// TIA Portal project "Project_Benzinarie" (V15.1)

(* hardware
DEVICE "S71500/ET200MP station_1"  S7-1500 station
   slot 0: "Rail_0"  Rack  6ES7 590-1***0-0AA0
   slot 1: "PLC_1"  CPU 1513-1 PN  6ES7 513-1AL02-0AB0  V2.6
      slot 3: "CPU display_1"  6ES7591-1AA00-0AA0
DEVICE "HMI_1"  KTP900 Basic PN
   slot 0: "HMI_1"  KTP900 Basic PN  6AV2 123-2JB03-0AX0  15.1.0.0
   slot 1: "HMI_RT_1"  KTP900 Basic PN  6AV2 123-2JB03-0AX0  15.1.0.0
   slot 5: "HMI_1.IE_CP_1"  PROFINET Interface  15.0.1.0
      slot 1: "PROFINET Interface_1"  PROFINET Interface
         slot 1: "Port_1"  Port
*)

// ===== PLC "PLC_1"  CPU 1513-1 PN =====

VAR_GLOBAL   // PLC tag table "Default tag table"
   "Clock_Byte" AT %MB0 : Byte;
   "Clock_10Hz" AT %M0.0 : Bool;
   "Clock_5Hz" AT %M0.1 : Bool;
   "Clock_2.5Hz" AT %M0.2 : Bool;
   "Clock_2Hz" AT %M0.3 : Bool;
   "Clock_1.25Hz" AT %M0.4 : Bool;
   "Clock_1Hz" AT %M0.5 : Bool;
   "Clock_0.625Hz" AT %M0.6 : Bool;
   "Clock_0.5Hz" AT %M0.7 : Bool;
END_VAR

DATA_BLOCK "Alarme"   // DB1
{ S7_Optimized_Access := 'TRUE' }
VERSION : 0.1
   VAR
      alarme_gather : Word;
      alarme_vect : Array[0..15] of Bool;
   END_VAR
BEGIN
END_DATA_BLOCK

DATA_BLOCK "Avarii"   // DB2
{ S7_Optimized_Access := 'TRUE' }
VERSION : 0.1
   VAR
      esd : Bool;
      esd_btn : Bool;
      reset_esd : Bool;
      avarie_p1 : Bool;
      avarie_p2 : Bool;
      avarie_p3 : Bool;
      avarie_p4 : Bool;
      avarie_generala : Bool;
      reset_avarii : Bool;
      plata_general : Bool;
   END_VAR
BEGIN
END_DATA_BLOCK

DATA_BLOCK "Bazine"   // DB3
{ S7_Optimized_Access := 'TRUE' }
VERSION : 0.1
   VAR
      benzina_90 : Real;
      benzina_95 : Real;
      motorina : Real;
      motorina_premium : Real;
      "benzina_90_1/2" : Real;
      "benzina_95_1/2" : Real;
      "motorina_1/2" : Real;
      "motorina_premium_1/2" : Real;
      b90_gol : Bool;
      b95_gol : Bool;
      m_gol : Bool;
      m_p_gol : Bool;
      bazin_gol_general : Bool;
      nivel_benzina90 : Real;
      nivel_benzina95 : Real;
      nivel_motorina : Real;
      nivel_motorina_premium : Real;
   END_VAR
BEGIN
END_DATA_BLOCK

DATA_BLOCK "Pompa_benzian90"   // DB4
{ S7_Optimized_Access := 'TRUE' }
VERSION : 0.1
   VAR
      blocare : Bool;
      scoasa : Bool;
      start_clapeta : Bool;
      buton_plata : Bool;
      led_rosu : Bool;
      permisiune_start : Bool;
      index_pret : Real;
      cantitate : Real;
      plata_posibila : Bool;
      terminat : Bool;
      pret : Real;
      nivel_pompa : Real;
      permisiune_pompa : Bool;
      pune_inapoi : Bool;
   END_VAR
BEGIN
END_DATA_BLOCK

DATA_BLOCK "Pompa_benzina95"   // DB5
{ S7_Optimized_Access := 'TRUE' }
VERSION : 0.1
   VAR
      blocare : Bool;
      scoasa : Bool;
      start_clapeta : Bool;
      buton_plata : Bool;
      led_rosu : Bool;
      permisiune_start : Bool;
      index_pret : Real;
      cantitate : Real;
      plata_posibila : Bool;
      terminat : Bool;
      pret : Real;
      nivel_pompa : Real;
      permisiune_pompa : Bool;
      pune_inapoi : Bool;
   END_VAR
BEGIN
END_DATA_BLOCK

DATA_BLOCK "Pompa_motorina"   // DB6
{ S7_Optimized_Access := 'TRUE' }
VERSION : 0.1
   VAR
      blocare : Bool;
      scoasa : Bool;
      start_clapeta : Bool;
      buton_plata : Bool;
      led_rosu : Bool;
      permisiune_start : Bool;
      index_pret : Real;
      cantitate : Real;
      plata_posibila : Bool;
      terminat : Bool;
      pret : Real;
      nivel_pompa : Real;
      permisiune_pompa : Bool;
      pune_inapoi : Bool;
   END_VAR
BEGIN
END_DATA_BLOCK

DATA_BLOCK "Pompa_motorina_premium"   // DB7
{ S7_Optimized_Access := 'TRUE' }
VERSION : 0.1
   VAR
      blocare : Bool;
      scoasa : Bool;
      start_clapeta : Bool;
      buton_plata : Bool;
      led_rosu : Bool;
      permisiune_start : Bool;
      index_pret : Real;
      cantitate : Real;
      plata_posibila : Bool;
      terminat : Bool;
      pret : Real;
      nivel_pompa : Real;
      permisiune_pompa : Bool;
      pune_inapoi : Bool;
   END_VAR
BEGIN
END_DATA_BLOCK

DATA_BLOCK "Benzina90"   // DB8
{ S7_Optimized_Access := 'TRUE' }
VERSION : 0.1
// stored: InstanceOfName Pompa
"Pompa"
BEGIN
END_DATA_BLOCK

DATA_BLOCK "Benzina95"   // DB9
{ S7_Optimized_Access := 'TRUE' }
VERSION : 0.1
// stored: InstanceOfName Pompa
"Pompa"
BEGIN
END_DATA_BLOCK

DATA_BLOCK "Motorina"   // DB10
{ S7_Optimized_Access := 'TRUE' }
VERSION : 0.1
// stored: InstanceOfName Pompa
"Pompa"
BEGIN
END_DATA_BLOCK

DATA_BLOCK "Motorina_premium"   // DB11
{ S7_Optimized_Access := 'TRUE' }
VERSION : 0.1
// stored: InstanceOfName Pompa
"Pompa"
BEGIN
END_DATA_BLOCK

DATA_BLOCK "Butoane_umplere_bazine"   // DB13
{ S7_Optimized_Access := 'TRUE' }
VERSION : 0.1
   VAR
      btn_b90 : Bool;
      btn_b95 : Bool;
      btn_m : Bool;
      btn_m_p : Bool;
   END_VAR
BEGIN
END_DATA_BLOCK

DATA_BLOCK "Hysteresis_DB"   // DB16
{ S7_Optimized_Access := 'TRUE' }
VERSION : 0.1
// stored: InstanceOfName Hysteresis
"Hysteresis"
BEGIN
END_DATA_BLOCK

// folder: System blocks/Program resources

DATA_BLOCK "reset_esd"   // DB12
{ S7_Optimized_Access := 'TRUE' }
AUTHOR : Simatic
FAMILY : IEC
NAME : IEC_TMR
VERSION : 1.0
// stored: InstanceOfName IEC_TIMER
"IEC_TIMER"
BEGIN
END_DATA_BLOCK

DATA_BLOCK "reset_avarii"   // DB14
{ S7_Optimized_Access := 'TRUE' }
AUTHOR : Simatic
FAMILY : IEC
NAME : IEC_TMR
VERSION : 1.0
// stored: InstanceOfName IEC_TIMER
"IEC_TIMER"
BEGIN
END_DATA_BLOCK

DATA_BLOCK "reset_umplere_b90"   // DB17
{ S7_Optimized_Access := 'TRUE' }
AUTHOR : Simatic
FAMILY : IEC
NAME : IEC_TMR
VERSION : 1.0
// stored: InstanceOfName IEC_TIMER
"IEC_TIMER"
BEGIN
END_DATA_BLOCK

DATA_BLOCK "reset_umplere_b95"   // DB18
{ S7_Optimized_Access := 'TRUE' }
AUTHOR : Simatic
FAMILY : IEC
NAME : IEC_TMR
VERSION : 1.0
// stored: InstanceOfName IEC_TIMER
"IEC_TIMER"
BEGIN
END_DATA_BLOCK

DATA_BLOCK "reset_umplere_m"   // DB19
{ S7_Optimized_Access := 'TRUE' }
AUTHOR : Simatic
FAMILY : IEC
NAME : IEC_TMR
VERSION : 1.0
// stored: InstanceOfName IEC_TIMER
"IEC_TIMER"
BEGIN
END_DATA_BLOCK

DATA_BLOCK "reset_umplere_m_p"   // DB20
{ S7_Optimized_Access := 'TRUE' }
AUTHOR : Simatic
FAMILY : IEC
NAME : IEC_TMR
VERSION : 1.0
// stored: InstanceOfName IEC_TIMER
"IEC_TIMER"
BEGIN
END_DATA_BLOCK

// folder: (top level)

FUNCTION_BLOCK "Pompa"   // FB1, LAD
{ S7_Optimized_Access := 'TRUE' }
VERSION : 0.1
   VAR_INPUT
      blocare : Bool;
      esd : Bool;
      avarie_interna : Bool;
      bazin_gol : Bool;
   END_VAR
   VAR_OUTPUT
      pret : Real;
      terminat : Bool;
   END_VAR
   VAR_IN_OUT
      scoasa : Bool;
      start_clapeta : Bool;
      bazin : Real;
      buton_plata : Bool;
      led_rosu : Bool;
      permisiune_start : Bool;
      permisiune_pompa : Bool;
      pune_inapoi : Bool;
      index_pret : Real;
      cantitate : Real;
      plata_posibila : Bool;
      nivel_pompa : Real;
   END_VAR
   VAR
      re1 : Bool;
      re2 : Bool;
      re3 : Bool;
      led_intermitent : Bool;
      timer_reset_plata : TON_TIME;
      Hysteresis_Instance : "Hysteresis";
   END_VAR
   VAR_TEMP   // added for the SCL form of the ladder/FBD networks
      _w1 : Bool;
   END_VAR
BEGIN

REGION Network 1: permisiune de start
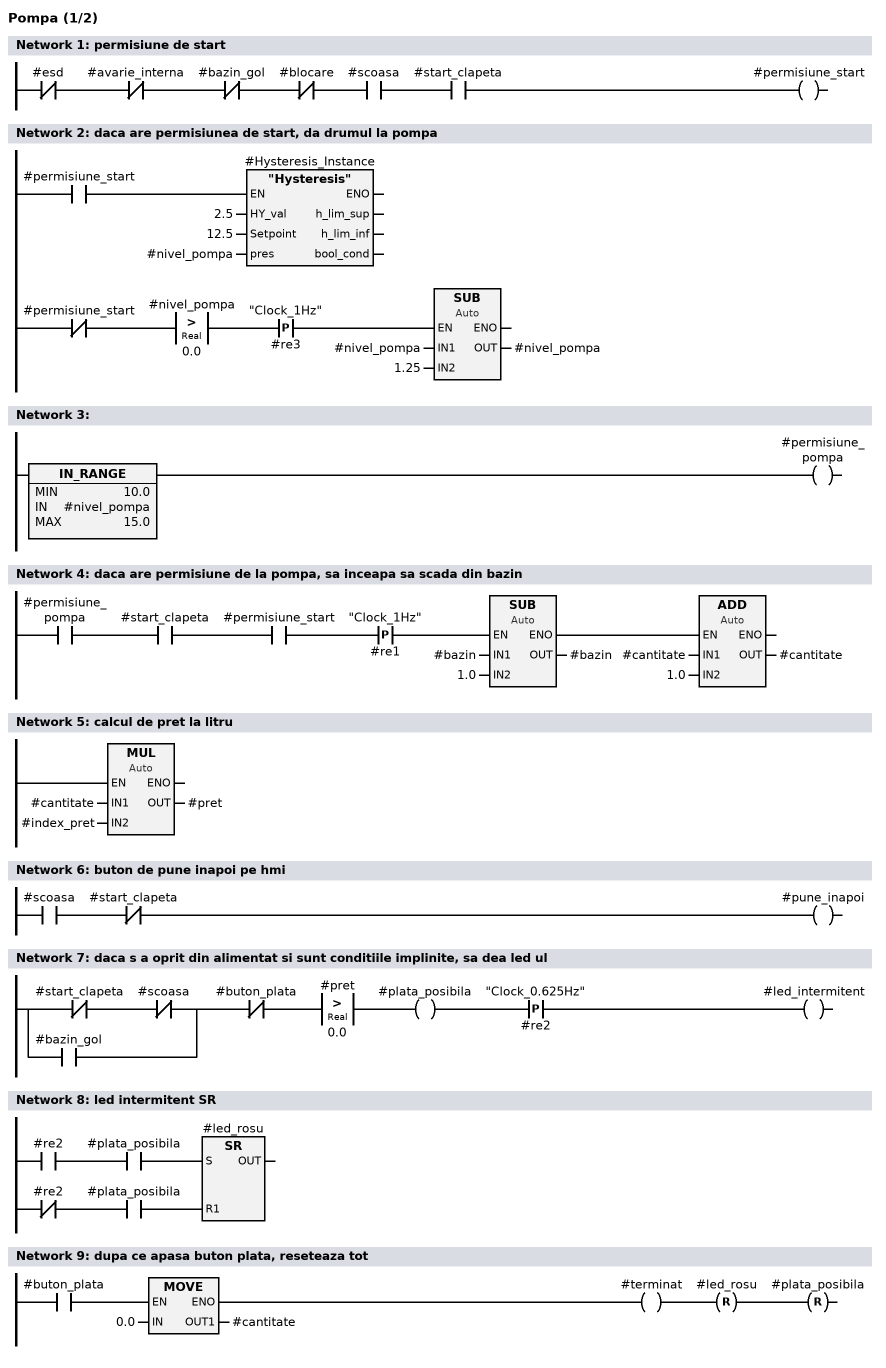
   RUNG wire#powerrail
      I_Contact( #esd )
      I_Contact( #avarie_interna )
      I_Contact( #bazin_gol )
      I_Contact( #blocare )
      Contact( #scoasa )
      Contact( #start_clapeta )
      Coil( #permisiune_start )
   END_RUNG
   // the same network as SCL:
   #permisiune_start := NOT #esd AND NOT #avarie_interna AND NOT #bazin_gol AND NOT #blocare AND #scoasa AND #start_clapeta;
END_REGION

REGION Network 2: daca are permisiunea de start, da drumul la pompa
   RUNG wire#powerrail
      Contact( #permisiune_start )
      #Hysteresis_Instance(HY_val := 2.5, Setpoint := 12.5, pres := #nivel_pompa, h_lim_sup =>, h_lim_inf =>, bool_cond =>)
   END_RUNG
   RUNG wire#powerrail
      I_Contact( #permisiune_start )
      { S7_Templates := "SrcType := Real" } GT_Contact(in1 := #nivel_pompa, in2 := 0.0)
      P_Contact(operand := "Clock_1Hz", bit := #re3)
      Sub(in1 := #nivel_pompa, in2 := 1.25, out => #nivel_pompa)
   END_RUNG
   // the same network as SCL:
   IF #permisiune_start THEN
       #Hysteresis_Instance(HY_val := 2.5, Setpoint := 12.5, pres := #nivel_pompa);   // "Hysteresis"
   END_IF;
   #_w1 := NOT #permisiune_start AND (#nivel_pompa > 0.0) AND "Clock_1Hz" AND NOT #re3;   // rising edge of "Clock_1Hz"
   #re3 := "Clock_1Hz";
   IF #_w1 THEN #nivel_pompa := #nivel_pompa - 1.25; END_IF;
END_REGION

REGION Network 3
   RUNG wire#powerrail
      { S7_Templates := "SrcType := Real" } InRange(min := 10.0, in := #nivel_pompa, max := 15.0)
      Coil( #permisiune_pompa )
   END_RUNG
   // the same network as SCL:
   #permisiune_pompa := (10.0 <= #nivel_pompa) AND (#nivel_pompa <= 15.0);
END_REGION

REGION Network 4: daca are permisiune de la pompa, sa inceapa sa scada din bazin
   RUNG wire#powerrail
      Contact( #permisiune_pompa )
      Contact( #start_clapeta )
      Contact( #permisiune_start )
      P_Contact(operand := "Clock_1Hz", bit := #re1)
      Sub(in1 := #bazin, in2 := 1.0, out => #bazin)
      Add(in1 := #cantitate, in2 := 1.0, out => #cantitate)
   END_RUNG
   // the same network as SCL:
   #_w1 := #permisiune_pompa AND #start_clapeta AND #permisiune_start AND "Clock_1Hz" AND NOT #re1;   // rising edge of "Clock_1Hz"
   #re1 := "Clock_1Hz";
   IF #_w1 THEN
       #bazin := #bazin - 1.0;
       #cantitate := #cantitate + 1.0;
   END_IF;
END_REGION

REGION Network 5: calcul de pret la litru
   RUNG wire#powerrail
      Mul(in1 := #cantitate, in2 := #index_pret, out => #pret)
   END_RUNG
   // the same network as SCL:
   #pret := #cantitate * #index_pret;
END_REGION

REGION Network 6: buton de pune inapoi pe hmi
   RUNG wire#powerrail
      Contact( #scoasa )
      I_Contact( #start_clapeta )
      Coil( #pune_inapoi )
   END_RUNG
   // the same network as SCL:
   #pune_inapoi := #scoasa AND NOT #start_clapeta;
END_REGION

REGION Network 7: daca s a oprit din alimentat si sunt conditiile implinite, sa dea led ul
   RUNG wire#powerrail
      I_Contact( #start_clapeta )
      I_Contact( #scoasa )
      wire#w1
      I_Contact( #buton_plata )
      { S7_Templates := "SrcType := Real" } GT_Contact(in1 := #pret, in2 := 0.0)
      Coil( #plata_posibila )
      P_Contact(operand := "Clock_0.625Hz", bit := #re2)
      Coil( #led_intermitent )
   END_RUNG
   RUNG wire#powerrail
      Contact( #bazin_gol )
   END_RUNG wire#w1
   // the same network as SCL:
   #plata_posibila := ((NOT #start_clapeta AND NOT #scoasa) OR #bazin_gol) AND NOT #buton_plata AND (#pret > 0.0);
   #_w1 := #plata_posibila AND "Clock_0.625Hz" AND NOT #re2;   // rising edge of "Clock_0.625Hz"
   #re2 := "Clock_0.625Hz";
   #led_intermitent := #_w1;
END_REGION

REGION Network 8: led intermitent SR
   RUNG wire#powerrail
      Contact( #re2 )
      Contact( #plata_posibila )
      S_SR(operand := #led_rosu, r1 := wire#w1)
   END_RUNG
   RUNG wire#powerrail
      I_Contact( #re2 )
      Contact( #plata_posibila )
   END_RUNG wire#w1
   // the same network as SCL:
   IF #re2 AND #plata_posibila THEN
       #led_rosu := TRUE;   // SR flip-flop
   END_IF;
   IF NOT #re2 AND #plata_posibila THEN #led_rosu := FALSE; END_IF;
END_REGION

REGION Network 9: dupa ce apasa buton plata, reseteaza tot
   RUNG wire#powerrail
      Contact( #buton_plata )
      Move(in := 0.0, out1 => #cantitate)
      Coil( #terminat )
      R_Coil( #led_rosu )
      R_Coil( #plata_posibila )
   END_RUNG
   // the same network as SCL:
   IF #buton_plata THEN #cantitate := 0.0; END_IF;
   #terminat := #buton_plata;
   IF #buton_plata THEN
       #led_rosu := FALSE;
       #plata_posibila := FALSE;
   END_IF;
END_REGION

REGION Network 10: reseteaza buton plata dupa 3 secunde
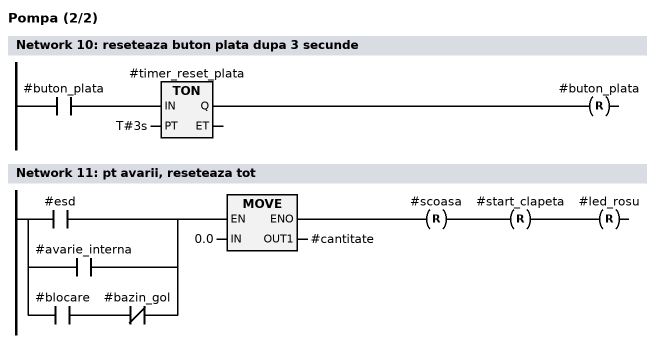
   #timer_reset_plata(IN := #buton_plata, PT := T#3s);   // TON
   IF #timer_reset_plata.Q THEN #buton_plata := FALSE; END_IF;
END_REGION

REGION Network 11: pt avarii, reseteaza tot
   RUNG wire#powerrail
      Contact( #esd )
      wire#w1
      Move(in := 0.0, out1 => #cantitate)
      R_Coil( #scoasa )
      R_Coil( #start_clapeta )
      R_Coil( #led_rosu )
   END_RUNG
   RUNG wire#powerrail
      Contact( #avarie_interna )
   END_RUNG wire#w1
   RUNG wire#powerrail
      Contact( #blocare )
      I_Contact( #bazin_gol )
   END_RUNG wire#w1
   // the same network as SCL:
   IF #esd OR #avarie_interna OR (#blocare AND NOT #bazin_gol) THEN
       #cantitate := 0.0;
       #scoasa := FALSE;
       #start_clapeta := FALSE;
       #led_rosu := FALSE;
   END_IF;
END_REGION
END_FUNCTION_BLOCK

FUNCTION_BLOCK "Hysteresis"   // FB2, LAD
{ S7_Optimized_Access := 'TRUE' }
VERSION : 0.1
   VAR_INPUT
      HY_val : Real;
      Setpoint : Real;
   END_VAR
   VAR_OUTPUT
      h_lim_sup : Real;
      h_lim_inf : Real;
      bool_cond : Bool;
   END_VAR
   VAR_IN_OUT
      pres : Real;
   END_VAR
   VAR
      re1 : Bool;
      re2 : Bool;
      urcare : Bool;
   END_VAR
   VAR_TEMP   // added for the SCL form of the ladder/FBD networks
      _w1 : Bool;
   END_VAR
BEGIN

REGION Network 1: daca are comanda de bool, sa creasca
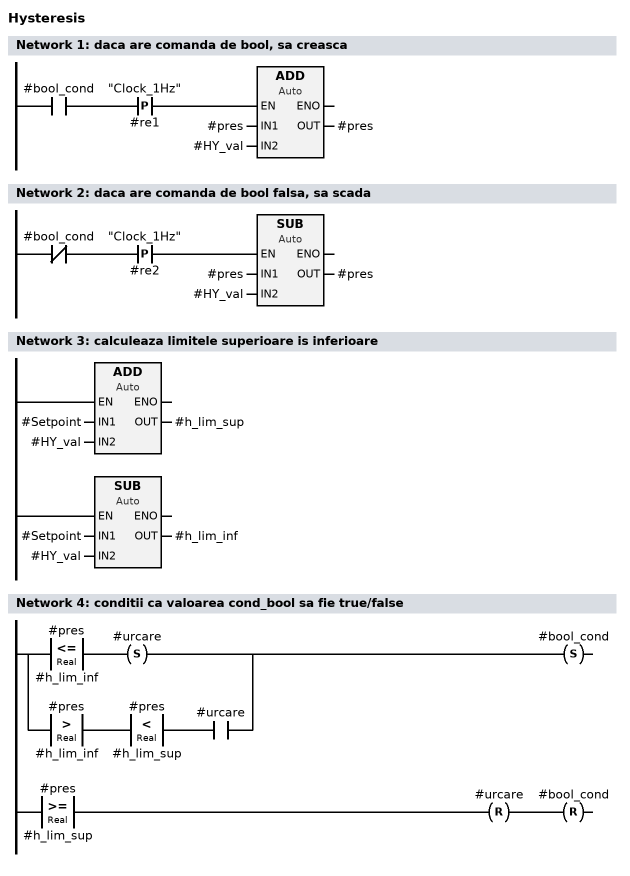
   RUNG wire#powerrail
      Contact( #bool_cond )
      P_Contact(operand := "Clock_1Hz", bit := #re1)
      Add(in1 := #pres, in2 := #HY_val, out => #pres)
   END_RUNG
   // the same network as SCL:
   #_w1 := #bool_cond AND "Clock_1Hz" AND NOT #re1;   // rising edge of "Clock_1Hz"
   #re1 := "Clock_1Hz";
   IF #_w1 THEN #pres := #pres + #HY_val; END_IF;
END_REGION

REGION Network 2: daca are comanda de bool falsa, sa scada
   RUNG wire#powerrail
      I_Contact( #bool_cond )
      P_Contact(operand := "Clock_1Hz", bit := #re2)
      Sub(in1 := #pres, in2 := #HY_val, out => #pres)
   END_RUNG
   // the same network as SCL:
   #_w1 := NOT #bool_cond AND "Clock_1Hz" AND NOT #re2;   // rising edge of "Clock_1Hz"
   #re2 := "Clock_1Hz";
   IF #_w1 THEN #pres := #pres - #HY_val; END_IF;
END_REGION

REGION Network 3: calculeaza limitele superioare is inferioare
   RUNG wire#powerrail
      Add(in1 := #Setpoint, in2 := #HY_val, out => #h_lim_sup)
   END_RUNG
   RUNG wire#powerrail
      Sub(in1 := #Setpoint, in2 := #HY_val, out => #h_lim_inf)
   END_RUNG
   // the same network as SCL:
   #h_lim_sup := #Setpoint + #HY_val;
   #h_lim_inf := #Setpoint - #HY_val;
END_REGION

REGION Network 4: conditii ca valoarea cond_bool sa fie true/false
   RUNG wire#powerrail
      { S7_Templates := "SrcType := Real" } LE_Contact(in1 := #pres, in2 := #h_lim_inf)
      S_Coil( #urcare )
      wire#w1
      S_Coil( #bool_cond )
   END_RUNG
   RUNG wire#powerrail
      { S7_Templates := "SrcType := Real" } GT_Contact(in1 := #pres, in2 := #h_lim_inf)
      { S7_Templates := "SrcType := Real" } LT_Contact(in1 := #pres, in2 := #h_lim_sup)
      Contact( #urcare )
   END_RUNG wire#w1
   RUNG wire#powerrail
      { S7_Templates := "SrcType := Real" } GE_Contact(in1 := #pres, in2 := #h_lim_sup)
      R_Coil( #urcare )
      R_Coil( #bool_cond )
   END_RUNG
   // the same network as SCL:
   #_w1 := #pres <= #h_lim_inf;
   IF #_w1 THEN #urcare := TRUE; END_IF;
   IF #_w1 OR ((#pres > #h_lim_inf) AND (#pres < #h_lim_sup) AND #urcare) THEN #bool_cond := TRUE; END_IF;
   IF #pres >= #h_lim_sup THEN
       #urcare := FALSE;
       #bool_cond := FALSE;
   END_IF;
END_REGION
END_FUNCTION_BLOCK

ORGANIZATION_BLOCK "Main"   // OB1, LAD, ProgramCycle
TITLE = "Main Program Sweep (Cycle)"
{ S7_Optimized_Access := 'TRUE' }
VERSION : 0.1
   VAR_INPUT
      Initial_Call : Bool;   // Initial call of this OB
      Remanence : Bool;   // =True, if remanent data are available
   END_VAR
   VAR_TEMP   // added for the SCL form of the ladder/FBD networks
      _w1 : Bool;
      _w2 : Bool;
      _w3 : Bool;
      _w4 : Bool;
   END_VAR
BEGIN

REGION Network 1: benzina90
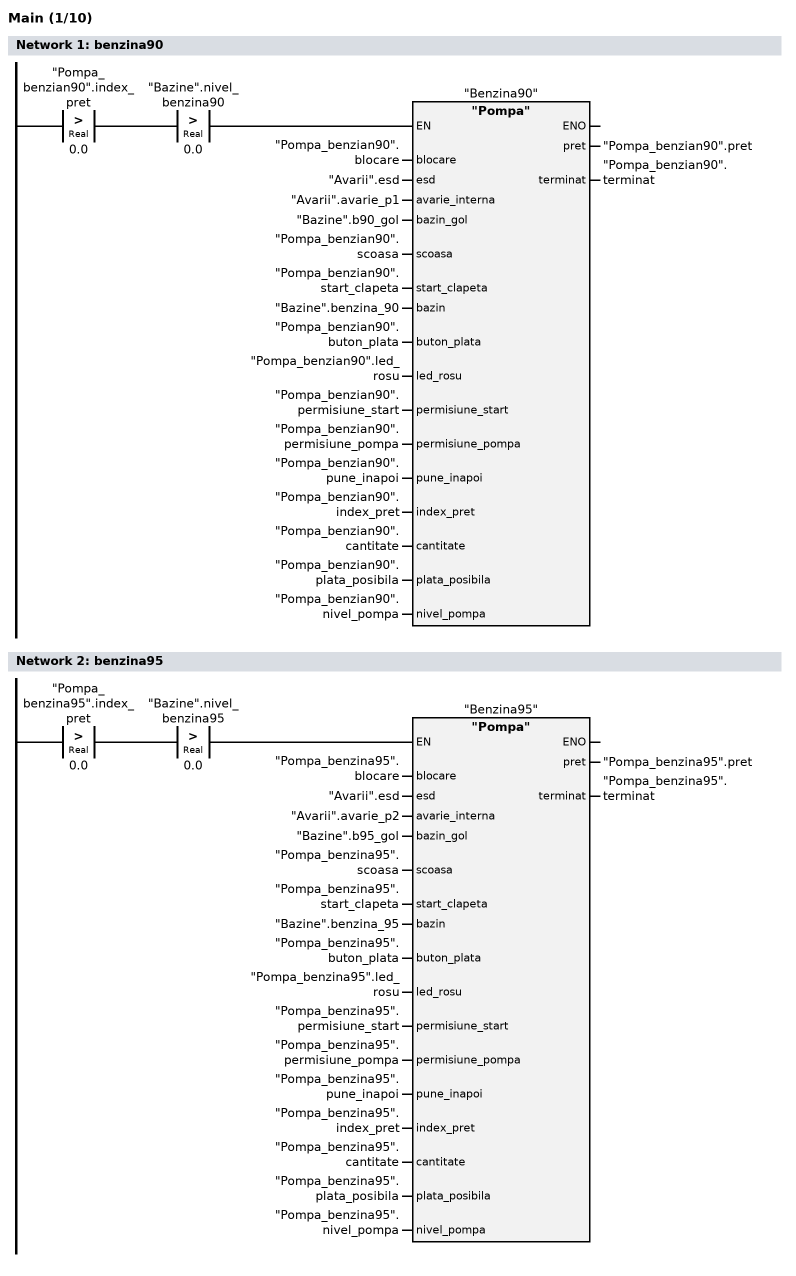
   RUNG wire#powerrail
      { S7_Templates := "SrcType := Real" } GT_Contact(in1 := "Pompa_benzian90".index_pret, in2 := 0.0)
      { S7_Templates := "SrcType := Real" } GT_Contact(in1 := "Bazine".nivel_benzina90, in2 := 0.0)
      "Benzina90"(blocare := "Pompa_benzian90".blocare, esd := "Avarii".esd, avarie_interna := "Avarii".avarie_p1, bazin_gol := "Bazine".b90_gol, scoasa := "Pompa_benzian90".scoasa, start_clapeta := "Pompa_benzian90".start_clapeta, bazin := "Bazine".benzina_90, buton_plata := "Pompa_benzian90".buton_plata, led_rosu := "Pompa_benzian90".led_rosu, permisiune_start := "Pompa_benzian90".permisiune_start, permisiune_pompa := "Pompa_benzian90".permisiune_pompa, pune_inapoi := "Pompa_benzian90".pune_inapoi, index_pret := "Pompa_benzian90".index_pret, cantitate := "Pompa_benzian90".cantitate, plata_posibila := "Pompa_benzian90".plata_posibila, nivel_pompa := "Pompa_benzian90".nivel_pompa, pret => "Pompa_benzian90".pret, terminat => "Pompa_benzian90".terminat)
   END_RUNG
   // the same network as SCL:
   IF ("Pompa_benzian90".index_pret > 0.0) AND ("Bazine".nivel_benzina90 > 0.0) THEN
       "Benzina90"(blocare := "Pompa_benzian90".blocare,   // "Pompa"
                   esd := "Avarii".esd,
                   avarie_interna := "Avarii".avarie_p1,
                   bazin_gol := "Bazine".b90_gol,
                   scoasa := "Pompa_benzian90".scoasa,
                   start_clapeta := "Pompa_benzian90".start_clapeta,
                   bazin := "Bazine".benzina_90,
                   buton_plata := "Pompa_benzian90".buton_plata,
                   led_rosu := "Pompa_benzian90".led_rosu,
                   permisiune_start := "Pompa_benzian90".permisiune_start,
                   permisiune_pompa := "Pompa_benzian90".permisiune_pompa,
                   pune_inapoi := "Pompa_benzian90".pune_inapoi,
                   index_pret := "Pompa_benzian90".index_pret,
                   cantitate := "Pompa_benzian90".cantitate,
                   plata_posibila := "Pompa_benzian90".plata_posibila,
                   nivel_pompa := "Pompa_benzian90".nivel_pompa,
                   pret => "Pompa_benzian90".pret,
                   terminat => "Pompa_benzian90".terminat);
   END_IF;
END_REGION

REGION Network 2: benzina95
   RUNG wire#powerrail
      { S7_Templates := "SrcType := Real" } GT_Contact(in1 := "Pompa_benzina95".index_pret, in2 := 0.0)
      { S7_Templates := "SrcType := Real" } GT_Contact(in1 := "Bazine".nivel_benzina95, in2 := 0.0)
      "Benzina95"(blocare := "Pompa_benzina95".blocare, esd := "Avarii".esd, avarie_interna := "Avarii".avarie_p2, bazin_gol := "Bazine".b95_gol, scoasa := "Pompa_benzina95".scoasa, start_clapeta := "Pompa_benzina95".start_clapeta, bazin := "Bazine".benzina_95, buton_plata := "Pompa_benzina95".buton_plata, led_rosu := "Pompa_benzina95".led_rosu, permisiune_start := "Pompa_benzina95".permisiune_start, permisiune_pompa := "Pompa_benzina95".permisiune_pompa, pune_inapoi := "Pompa_benzina95".pune_inapoi, index_pret := "Pompa_benzina95".index_pret, cantitate := "Pompa_benzina95".cantitate, plata_posibila := "Pompa_benzina95".plata_posibila, nivel_pompa := "Pompa_benzina95".nivel_pompa, pret => "Pompa_benzina95".pret, terminat => "Pompa_benzina95".terminat)
   END_RUNG
   // the same network as SCL:
   IF ("Pompa_benzina95".index_pret > 0.0) AND ("Bazine".nivel_benzina95 > 0.0) THEN
       "Benzina95"(blocare := "Pompa_benzina95".blocare,   // "Pompa"
                   esd := "Avarii".esd,
                   avarie_interna := "Avarii".avarie_p2,
                   bazin_gol := "Bazine".b95_gol,
                   scoasa := "Pompa_benzina95".scoasa,
                   start_clapeta := "Pompa_benzina95".start_clapeta,
                   bazin := "Bazine".benzina_95,
                   buton_plata := "Pompa_benzina95".buton_plata,
                   led_rosu := "Pompa_benzina95".led_rosu,
                   permisiune_start := "Pompa_benzina95".permisiune_start,
                   permisiune_pompa := "Pompa_benzina95".permisiune_pompa,
                   pune_inapoi := "Pompa_benzina95".pune_inapoi,
                   index_pret := "Pompa_benzina95".index_pret,
                   cantitate := "Pompa_benzina95".cantitate,
                   plata_posibila := "Pompa_benzina95".plata_posibila,
                   nivel_pompa := "Pompa_benzina95".nivel_pompa,
                   pret => "Pompa_benzina95".pret,
                   terminat => "Pompa_benzina95".terminat);
   END_IF;
END_REGION

REGION Network 3: motorina
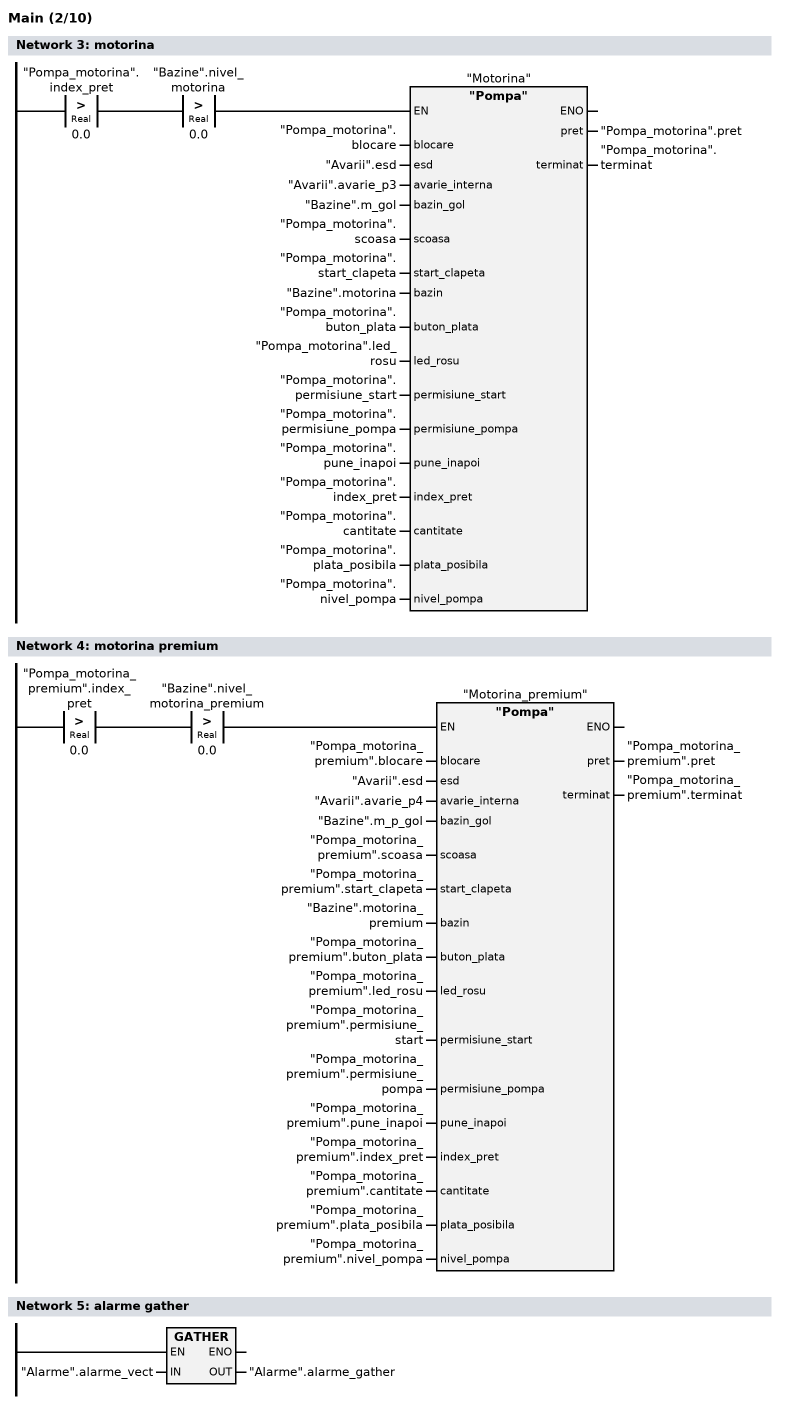
   RUNG wire#powerrail
      { S7_Templates := "SrcType := Real" } GT_Contact(in1 := "Pompa_motorina".index_pret, in2 := 0.0)
      { S7_Templates := "SrcType := Real" } GT_Contact(in1 := "Bazine".nivel_motorina, in2 := 0.0)
      "Motorina"(blocare := "Pompa_motorina".blocare, esd := "Avarii".esd, avarie_interna := "Avarii".avarie_p3, bazin_gol := "Bazine".m_gol, scoasa := "Pompa_motorina".scoasa, start_clapeta := "Pompa_motorina".start_clapeta, bazin := "Bazine".motorina, buton_plata := "Pompa_motorina".buton_plata, led_rosu := "Pompa_motorina".led_rosu, permisiune_start := "Pompa_motorina".permisiune_start, permisiune_pompa := "Pompa_motorina".permisiune_pompa, pune_inapoi := "Pompa_motorina".pune_inapoi, index_pret := "Pompa_motorina".index_pret, cantitate := "Pompa_motorina".cantitate, plata_posibila := "Pompa_motorina".plata_posibila, nivel_pompa := "Pompa_motorina".nivel_pompa, pret => "Pompa_motorina".pret, terminat => "Pompa_motorina".terminat)
   END_RUNG
   // the same network as SCL:
   IF ("Pompa_motorina".index_pret > 0.0) AND ("Bazine".nivel_motorina > 0.0) THEN
       "Motorina"(blocare := "Pompa_motorina".blocare,   // "Pompa"
                  esd := "Avarii".esd,
                  avarie_interna := "Avarii".avarie_p3,
                  bazin_gol := "Bazine".m_gol,
                  scoasa := "Pompa_motorina".scoasa,
                  start_clapeta := "Pompa_motorina".start_clapeta,
                  bazin := "Bazine".motorina,
                  buton_plata := "Pompa_motorina".buton_plata,
                  led_rosu := "Pompa_motorina".led_rosu,
                  permisiune_start := "Pompa_motorina".permisiune_start,
                  permisiune_pompa := "Pompa_motorina".permisiune_pompa,
                  pune_inapoi := "Pompa_motorina".pune_inapoi,
                  index_pret := "Pompa_motorina".index_pret,
                  cantitate := "Pompa_motorina".cantitate,
                  plata_posibila := "Pompa_motorina".plata_posibila,
                  nivel_pompa := "Pompa_motorina".nivel_pompa,
                  pret => "Pompa_motorina".pret,
                  terminat => "Pompa_motorina".terminat);
   END_IF;
END_REGION

REGION Network 4: motorina premium
   RUNG wire#powerrail
      { S7_Templates := "SrcType := Real" } GT_Contact(in1 := "Pompa_motorina_premium".index_pret, in2 := 0.0)
      { S7_Templates := "SrcType := Real" } GT_Contact(in1 := "Bazine".nivel_motorina_premium, in2 := 0.0)
      "Motorina_premium"(blocare := "Pompa_motorina_premium".blocare, esd := "Avarii".esd, avarie_interna := "Avarii".avarie_p4, bazin_gol := "Bazine".m_p_gol, scoasa := "Pompa_motorina_premium".scoasa, start_clapeta := "Pompa_motorina_premium".start_clapeta, bazin := "Bazine".motorina_premium, buton_plata := "Pompa_motorina_premium".buton_plata, led_rosu := "Pompa_motorina_premium".led_rosu, permisiune_start := "Pompa_motorina_premium".permisiune_start, permisiune_pompa := "Pompa_motorina_premium".permisiune_pompa, pune_inapoi := "Pompa_motorina_premium".pune_inapoi, index_pret := "Pompa_motorina_premium".index_pret, cantitate := "Pompa_motorina_premium".cantitate, plata_posibila := "Pompa_motorina_premium".plata_posibila, nivel_pompa := "Pompa_motorina_premium".nivel_pompa, pret => "Pompa_motorina_premium".pret, terminat => "Pompa_motorina_premium".terminat)
   END_RUNG
   // the same network as SCL:
   IF ("Pompa_motorina_premium".index_pret > 0.0) AND ("Bazine".nivel_motorina_premium > 0.0) THEN
       "Motorina_premium"(blocare := "Pompa_motorina_premium".blocare,   // "Pompa"
                          esd := "Avarii".esd,
                          avarie_interna := "Avarii".avarie_p4,
                          bazin_gol := "Bazine".m_p_gol,
                          scoasa := "Pompa_motorina_premium".scoasa,
                          start_clapeta := "Pompa_motorina_premium".start_clapeta,
                          bazin := "Bazine".motorina_premium,
                          buton_plata := "Pompa_motorina_premium".buton_plata,
                          led_rosu := "Pompa_motorina_premium".led_rosu,
                          permisiune_start := "Pompa_motorina_premium".permisiune_start,
                          permisiune_pompa := "Pompa_motorina_premium".permisiune_pompa,
                          pune_inapoi := "Pompa_motorina_premium".pune_inapoi,
                          index_pret := "Pompa_motorina_premium".index_pret,
                          cantitate := "Pompa_motorina_premium".cantitate,
                          plata_posibila := "Pompa_motorina_premium".plata_posibila,
                          nivel_pompa := "Pompa_motorina_premium".nivel_pompa,
                          pret => "Pompa_motorina_premium".pret,
                          terminat => "Pompa_motorina_premium".terminat);
   END_IF;
END_REGION

REGION Network 5: alarme gather
   GATHER(IN := "Alarme".alarme_vect, OUT => "Alarme".alarme_gather);
END_REGION

REGION Network 6: umplere bazin la maxim cand e apasat butonul
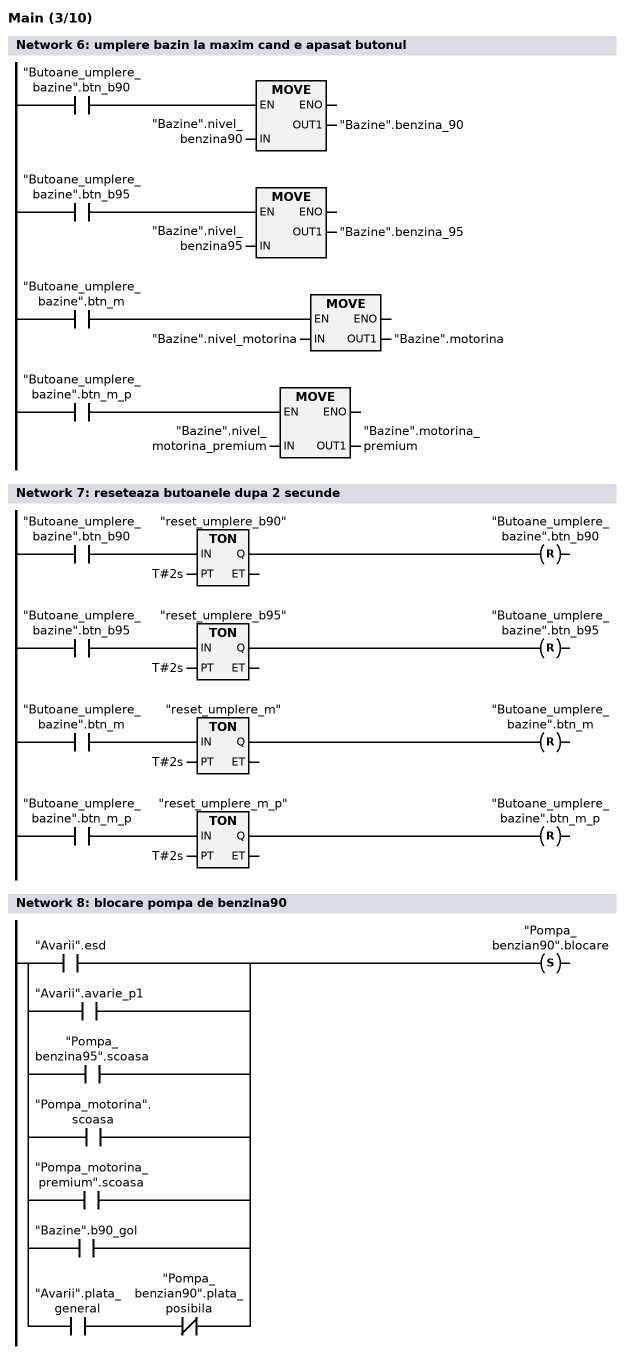
   RUNG wire#powerrail
      Contact( "Butoane_umplere_bazine".btn_b90 )
      Move(in := "Bazine".nivel_benzina90, out1 => "Bazine".benzina_90)
   END_RUNG
   RUNG wire#powerrail
      Contact( "Butoane_umplere_bazine".btn_b95 )
      Move(in := "Bazine".nivel_benzina95, out1 => "Bazine".benzina_95)
   END_RUNG
   RUNG wire#powerrail
      Contact( "Butoane_umplere_bazine".btn_m )
      Move(in := "Bazine".nivel_motorina, out1 => "Bazine".motorina)
   END_RUNG
   RUNG wire#powerrail
      Contact( "Butoane_umplere_bazine".btn_m_p )
      Move(in := "Bazine".nivel_motorina_premium, out1 => "Bazine".motorina_premium)
   END_RUNG
   // the same network as SCL:
   IF "Butoane_umplere_bazine".btn_b90 THEN "Bazine".benzina_90 := "Bazine".nivel_benzina90; END_IF;
   IF "Butoane_umplere_bazine".btn_b95 THEN "Bazine".benzina_95 := "Bazine".nivel_benzina95; END_IF;
   IF "Butoane_umplere_bazine".btn_m THEN "Bazine".motorina := "Bazine".nivel_motorina; END_IF;
   IF "Butoane_umplere_bazine".btn_m_p THEN
       "Bazine".motorina_premium := "Bazine".nivel_motorina_premium;
   END_IF;
END_REGION

REGION Network 7: reseteaza butoanele dupa 2 secunde
   "reset_umplere_b90".TON(IN := "Butoane_umplere_bazine".btn_b90, PT := T#2s);
   IF "reset_umplere_b90".Q THEN "Butoane_umplere_bazine".btn_b90 := FALSE; END_IF;
   "reset_umplere_b95".TON(IN := "Butoane_umplere_bazine".btn_b95, PT := T#2s);
   IF "reset_umplere_b95".Q THEN "Butoane_umplere_bazine".btn_b95 := FALSE; END_IF;
   "reset_umplere_m".TON(IN := "Butoane_umplere_bazine".btn_m, PT := T#2s);
   IF "reset_umplere_m".Q THEN "Butoane_umplere_bazine".btn_m := FALSE; END_IF;
   "reset_umplere_m_p".TON(IN := "Butoane_umplere_bazine".btn_m_p, PT := T#2s);
   IF "reset_umplere_m_p".Q THEN "Butoane_umplere_bazine".btn_m_p := FALSE; END_IF;
END_REGION

REGION Network 8: blocare pompa de benzina90
   RUNG wire#powerrail
      Contact( "Avarii".esd )
      wire#w1
      S_Coil( "Pompa_benzian90".blocare )
   END_RUNG
   RUNG wire#powerrail
      Contact( "Avarii".avarie_p1 )
   END_RUNG wire#w1
   RUNG wire#powerrail
      Contact( "Pompa_benzina95".scoasa )
   END_RUNG wire#w1
   RUNG wire#powerrail
      Contact( "Pompa_motorina".scoasa )
   END_RUNG wire#w1
   RUNG wire#powerrail
      Contact( "Pompa_motorina_premium".scoasa )
   END_RUNG wire#w1
   RUNG wire#powerrail
      Contact( "Bazine".b90_gol )
   END_RUNG wire#w1
   RUNG wire#powerrail
      Contact( "Avarii".plata_general )
      I_Contact( "Pompa_benzian90".plata_posibila )
   END_RUNG wire#w1
   // the same network as SCL:
   IF "Avarii".esd OR "Avarii".avarie_p1 OR "Pompa_benzina95".scoasa OR "Pompa_motorina".scoasa OR "Pompa_motorina_premium".scoasa OR "Bazine".b90_gol OR ("Avarii".plata_general AND NOT "Pompa_benzian90".plata_posibila) THEN
       "Pompa_benzian90".blocare := TRUE;
   END_IF;
END_REGION

REGION Network 9: blocare pompa de benzina95
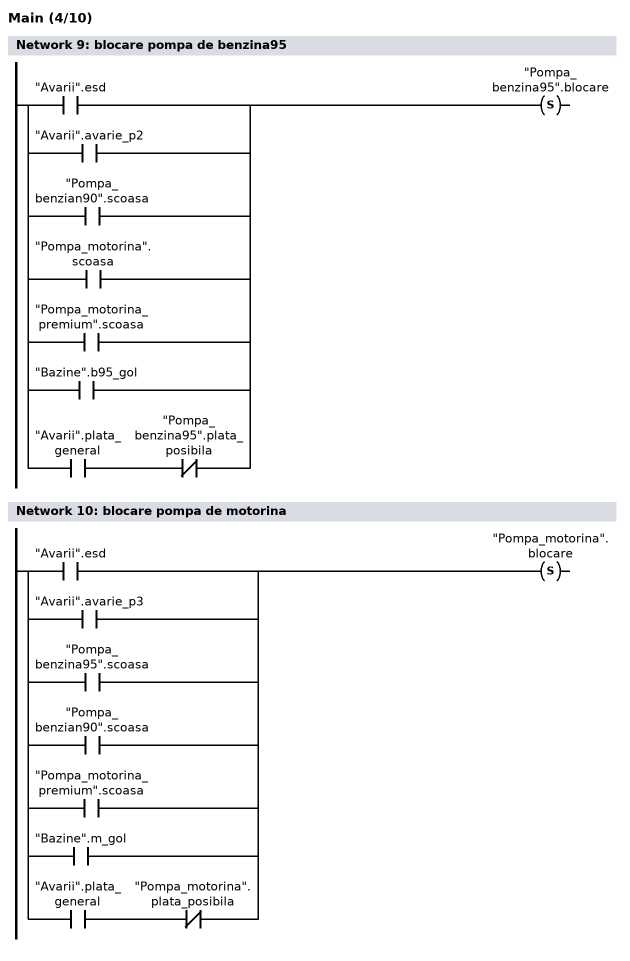
   RUNG wire#powerrail
      Contact( "Avarii".esd )
      wire#w1
      S_Coil( "Pompa_benzina95".blocare )
   END_RUNG
   RUNG wire#powerrail
      Contact( "Avarii".avarie_p2 )
   END_RUNG wire#w1
   RUNG wire#powerrail
      Contact( "Pompa_benzian90".scoasa )
   END_RUNG wire#w1
   RUNG wire#powerrail
      Contact( "Pompa_motorina".scoasa )
   END_RUNG wire#w1
   RUNG wire#powerrail
      Contact( "Pompa_motorina_premium".scoasa )
   END_RUNG wire#w1
   RUNG wire#powerrail
      Contact( "Bazine".b95_gol )
   END_RUNG wire#w1
   RUNG wire#powerrail
      Contact( "Avarii".plata_general )
      I_Contact( "Pompa_benzina95".plata_posibila )
   END_RUNG wire#w1
   // the same network as SCL:
   IF "Avarii".esd OR "Avarii".avarie_p2 OR "Pompa_benzian90".scoasa OR "Pompa_motorina".scoasa OR "Pompa_motorina_premium".scoasa OR "Bazine".b95_gol OR ("Avarii".plata_general AND NOT "Pompa_benzina95".plata_posibila) THEN
       "Pompa_benzina95".blocare := TRUE;
   END_IF;
END_REGION

REGION Network 10: blocare pompa de motorina
   RUNG wire#powerrail
      Contact( "Avarii".esd )
      wire#w1
      S_Coil( "Pompa_motorina".blocare )
   END_RUNG
   RUNG wire#powerrail
      Contact( "Avarii".avarie_p3 )
   END_RUNG wire#w1
   RUNG wire#powerrail
      Contact( "Pompa_benzina95".scoasa )
   END_RUNG wire#w1
   RUNG wire#powerrail
      Contact( "Pompa_benzian90".scoasa )
   END_RUNG wire#w1
   RUNG wire#powerrail
      Contact( "Pompa_motorina_premium".scoasa )
   END_RUNG wire#w1
   RUNG wire#powerrail
      Contact( "Bazine".m_gol )
   END_RUNG wire#w1
   RUNG wire#powerrail
      Contact( "Avarii".plata_general )
      I_Contact( "Pompa_motorina".plata_posibila )
   END_RUNG wire#w1
   // the same network as SCL:
   IF "Avarii".esd OR "Avarii".avarie_p3 OR "Pompa_benzina95".scoasa OR "Pompa_benzian90".scoasa OR "Pompa_motorina_premium".scoasa OR "Bazine".m_gol OR ("Avarii".plata_general AND NOT "Pompa_motorina".plata_posibila) THEN
       "Pompa_motorina".blocare := TRUE;
   END_IF;
END_REGION

REGION Network 11: blocare pompa de motorina premium
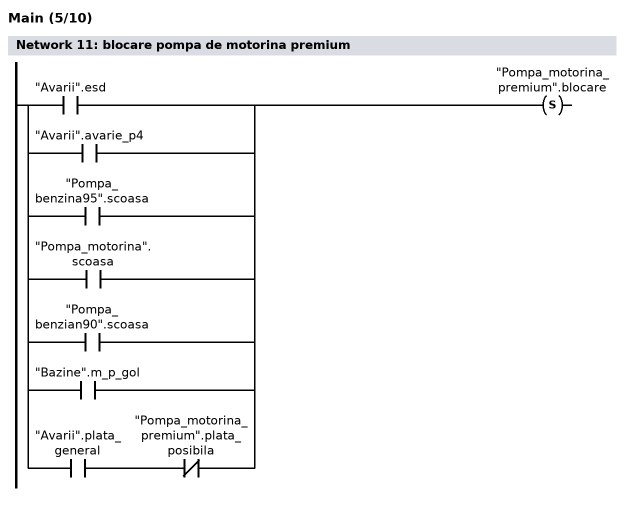
   RUNG wire#powerrail
      Contact( "Avarii".esd )
      wire#w1
      S_Coil( "Pompa_motorina_premium".blocare )
   END_RUNG
   RUNG wire#powerrail
      Contact( "Avarii".avarie_p4 )
   END_RUNG wire#w1
   RUNG wire#powerrail
      Contact( "Pompa_benzina95".scoasa )
   END_RUNG wire#w1
   RUNG wire#powerrail
      Contact( "Pompa_motorina".scoasa )
   END_RUNG wire#w1
   RUNG wire#powerrail
      Contact( "Pompa_benzian90".scoasa )
   END_RUNG wire#w1
   RUNG wire#powerrail
      Contact( "Bazine".m_p_gol )
   END_RUNG wire#w1
   RUNG wire#powerrail
      Contact( "Avarii".plata_general )
      I_Contact( "Pompa_motorina_premium".plata_posibila )
   END_RUNG wire#w1
   // the same network as SCL:
   IF "Avarii".esd OR "Avarii".avarie_p4 OR "Pompa_benzina95".scoasa OR "Pompa_motorina".scoasa OR "Pompa_benzian90".scoasa OR "Bazine".m_p_gol OR ("Avarii".plata_general AND NOT "Pompa_motorina_premium".plata_posibila) THEN
       "Pompa_motorina_premium".blocare := TRUE;
   END_IF;
END_REGION

REGION Network 12: reseteaza blocarea la pompe daca se termina
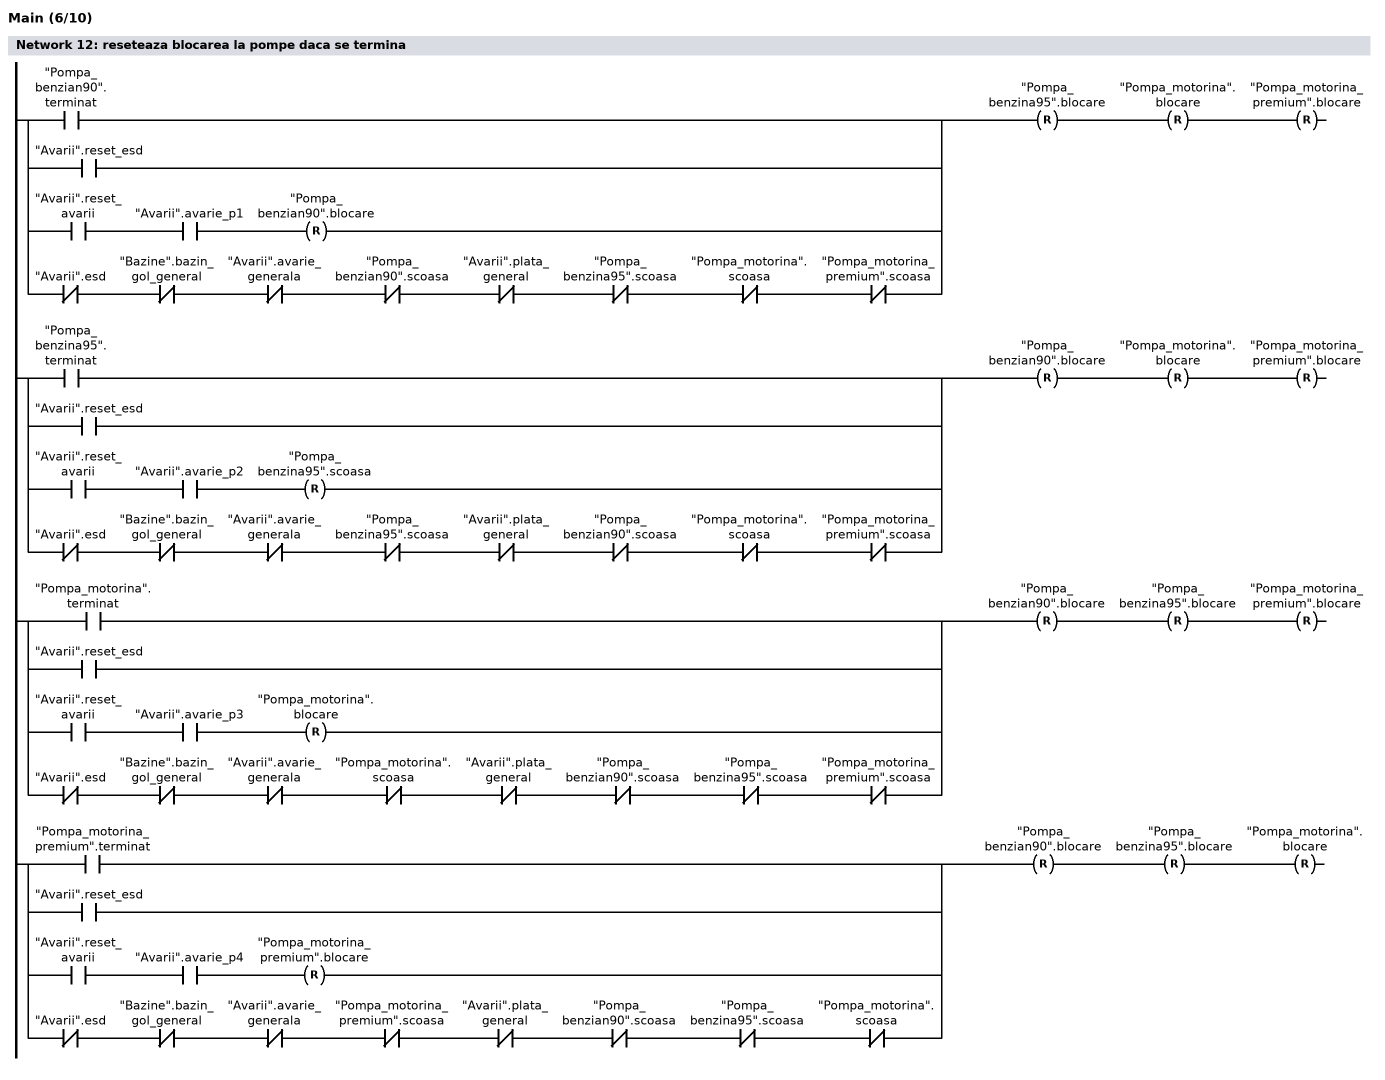
   RUNG wire#powerrail
      Contact( "Pompa_benzian90".terminat )
      wire#w1
      R_Coil( "Pompa_benzina95".blocare )
      R_Coil( "Pompa_motorina".blocare )
      R_Coil( "Pompa_motorina_premium".blocare )
   END_RUNG
   RUNG wire#powerrail
      Contact( "Avarii".reset_esd )
   END_RUNG wire#w1
   RUNG wire#powerrail
      Contact( "Avarii".reset_avarii )
      Contact( "Avarii".avarie_p1 )
      R_Coil( "Pompa_benzian90".blocare )
   END_RUNG wire#w1
   RUNG wire#powerrail
      I_Contact( "Avarii".esd )
      I_Contact( "Bazine".bazin_gol_general )
      I_Contact( "Avarii".avarie_generala )
      I_Contact( "Pompa_benzian90".scoasa )
      I_Contact( "Avarii".plata_general )
      I_Contact( "Pompa_benzina95".scoasa )
      I_Contact( "Pompa_motorina".scoasa )
      I_Contact( "Pompa_motorina_premium".scoasa )
   END_RUNG wire#w1
   RUNG wire#powerrail
      Contact( "Pompa_benzina95".terminat )
      wire#w2
      R_Coil( "Pompa_benzian90".blocare )
      R_Coil( "Pompa_motorina".blocare )
      R_Coil( "Pompa_motorina_premium".blocare )
   END_RUNG
   RUNG wire#powerrail
      Contact( "Avarii".reset_esd )
   END_RUNG wire#w2
   RUNG wire#powerrail
      Contact( "Avarii".reset_avarii )
      Contact( "Avarii".avarie_p2 )
      R_Coil( "Pompa_benzina95".scoasa )
   END_RUNG wire#w2
   RUNG wire#powerrail
      I_Contact( "Avarii".esd )
      I_Contact( "Bazine".bazin_gol_general )
      I_Contact( "Avarii".avarie_generala )
      I_Contact( "Pompa_benzina95".scoasa )
      I_Contact( "Avarii".plata_general )
      I_Contact( "Pompa_benzian90".scoasa )
      I_Contact( "Pompa_motorina".scoasa )
      I_Contact( "Pompa_motorina_premium".scoasa )
   END_RUNG wire#w2
   RUNG wire#powerrail
      Contact( "Pompa_motorina".terminat )
      wire#w3
      R_Coil( "Pompa_benzian90".blocare )
      R_Coil( "Pompa_benzina95".blocare )
      R_Coil( "Pompa_motorina_premium".blocare )
   END_RUNG
   RUNG wire#powerrail
      Contact( "Avarii".reset_esd )
   END_RUNG wire#w3
   RUNG wire#powerrail
      Contact( "Avarii".reset_avarii )
      Contact( "Avarii".avarie_p3 )
      R_Coil( "Pompa_motorina".blocare )
   END_RUNG wire#w3
   RUNG wire#powerrail
      I_Contact( "Avarii".esd )
      I_Contact( "Bazine".bazin_gol_general )
      I_Contact( "Avarii".avarie_generala )
      I_Contact( "Pompa_motorina".scoasa )
      I_Contact( "Avarii".plata_general )
      I_Contact( "Pompa_benzian90".scoasa )
      I_Contact( "Pompa_benzina95".scoasa )
      I_Contact( "Pompa_motorina_premium".scoasa )
   END_RUNG wire#w3
   RUNG wire#powerrail
      Contact( "Pompa_motorina_premium".terminat )
      wire#w4
      R_Coil( "Pompa_benzian90".blocare )
      R_Coil( "Pompa_benzina95".blocare )
      R_Coil( "Pompa_motorina".blocare )
   END_RUNG
   RUNG wire#powerrail
      Contact( "Avarii".reset_esd )
   END_RUNG wire#w4
   RUNG wire#powerrail
      Contact( "Avarii".reset_avarii )
      Contact( "Avarii".avarie_p4 )
      R_Coil( "Pompa_motorina_premium".blocare )
   END_RUNG wire#w4
   RUNG wire#powerrail
      I_Contact( "Avarii".esd )
      I_Contact( "Bazine".bazin_gol_general )
      I_Contact( "Avarii".avarie_generala )
      I_Contact( "Pompa_motorina_premium".scoasa )
      I_Contact( "Avarii".plata_general )
      I_Contact( "Pompa_benzian90".scoasa )
      I_Contact( "Pompa_benzina95".scoasa )
      I_Contact( "Pompa_motorina".scoasa )
   END_RUNG wire#w4
   // the same network as SCL:
   #_w1 := "Avarii".reset_avarii AND "Avarii".avarie_p1;
   IF #_w1 THEN "Pompa_benzian90".blocare := FALSE; END_IF;
   IF "Pompa_benzian90".terminat OR "Avarii".reset_esd OR #_w1 OR (NOT "Avarii".esd AND NOT "Bazine".bazin_gol_general AND NOT "Avarii".avarie_generala AND NOT "Pompa_benzian90".scoasa AND NOT "Avarii".plata_general AND NOT "Pompa_benzina95".scoasa AND NOT "Pompa_motorina".scoasa AND NOT "Pompa_motorina_premium".scoasa) THEN
       "Pompa_benzina95".blocare := FALSE;
       "Pompa_motorina".blocare := FALSE;
       "Pompa_motorina_premium".blocare := FALSE;
   END_IF;
   #_w2 := "Avarii".reset_avarii AND "Avarii".avarie_p2;
   IF #_w2 THEN "Pompa_benzina95".scoasa := FALSE; END_IF;
   IF "Pompa_benzina95".terminat OR "Avarii".reset_esd OR #_w2 OR (NOT "Avarii".esd AND NOT "Bazine".bazin_gol_general AND NOT "Avarii".avarie_generala AND NOT "Pompa_benzina95".scoasa AND NOT "Avarii".plata_general AND NOT "Pompa_benzian90".scoasa AND NOT "Pompa_motorina".scoasa AND NOT "Pompa_motorina_premium".scoasa) THEN
       "Pompa_benzian90".blocare := FALSE;
       "Pompa_motorina".blocare := FALSE;
       "Pompa_motorina_premium".blocare := FALSE;
   END_IF;
   #_w3 := "Avarii".reset_avarii AND "Avarii".avarie_p3;
   IF #_w3 THEN "Pompa_motorina".blocare := FALSE; END_IF;
   IF "Pompa_motorina".terminat OR "Avarii".reset_esd OR #_w3 OR (NOT "Avarii".esd AND NOT "Bazine".bazin_gol_general AND NOT "Avarii".avarie_generala AND NOT "Pompa_motorina".scoasa AND NOT "Avarii".plata_general AND NOT "Pompa_benzian90".scoasa AND NOT "Pompa_benzina95".scoasa AND NOT "Pompa_motorina_premium".scoasa) THEN
       "Pompa_benzian90".blocare := FALSE;
       "Pompa_benzina95".blocare := FALSE;
       "Pompa_motorina_premium".blocare := FALSE;
   END_IF;
   #_w4 := "Avarii".reset_avarii AND "Avarii".avarie_p4;
   IF #_w4 THEN "Pompa_motorina_premium".blocare := FALSE; END_IF;
   IF "Pompa_motorina_premium".terminat OR "Avarii".reset_esd OR #_w4 OR (NOT "Avarii".esd AND NOT "Bazine".bazin_gol_general AND NOT "Avarii".avarie_generala AND NOT "Pompa_motorina_premium".scoasa AND NOT "Avarii".plata_general AND NOT "Pompa_benzian90".scoasa AND NOT "Pompa_benzina95".scoasa AND NOT "Pompa_motorina".scoasa) THEN
       "Pompa_benzian90".blocare := FALSE;
       "Pompa_benzina95".blocare := FALSE;
       "Pompa_motorina".blocare := FALSE;
   END_IF;
END_REGION

REGION Network 13: calculeaza jumatatea bazinelor
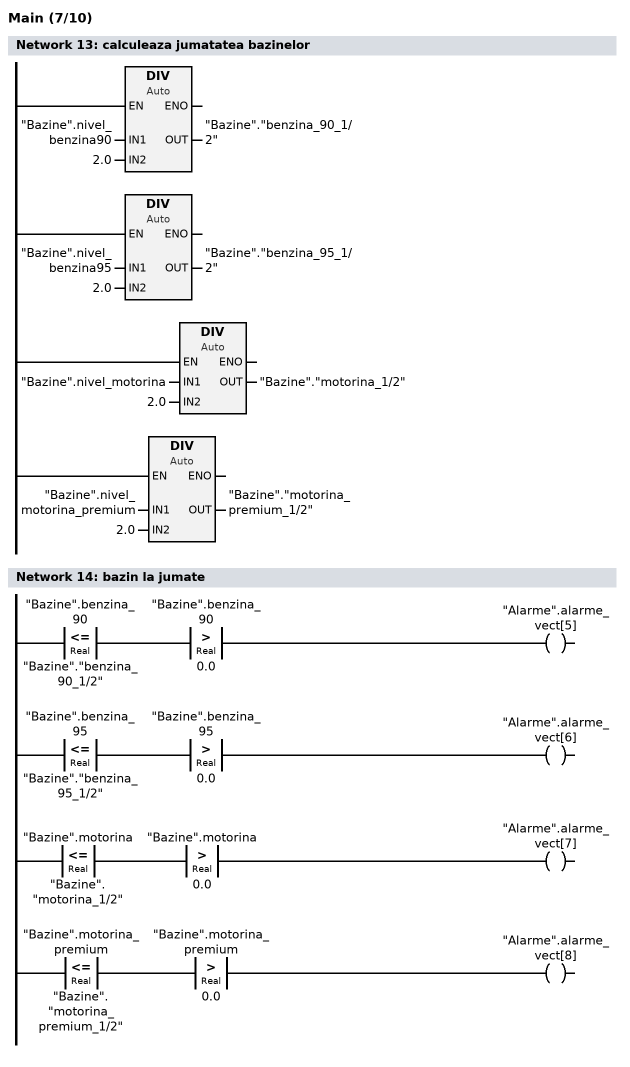
   RUNG wire#powerrail
      Div(in1 := "Bazine".nivel_benzina90, in2 := 2.0, out => "Bazine"."benzina_90_1/2")
   END_RUNG
   RUNG wire#powerrail
      Div(in1 := "Bazine".nivel_benzina95, in2 := 2.0, out => "Bazine"."benzina_95_1/2")
   END_RUNG
   RUNG wire#powerrail
      Div(in1 := "Bazine".nivel_motorina, in2 := 2.0, out => "Bazine"."motorina_1/2")
   END_RUNG
   RUNG wire#powerrail
      Div(in1 := "Bazine".nivel_motorina_premium, in2 := 2.0, out => "Bazine"."motorina_premium_1/2")
   END_RUNG
   // the same network as SCL:
   "Bazine"."benzina_90_1/2" := "Bazine".nivel_benzina90 / 2.0;
   "Bazine"."benzina_95_1/2" := "Bazine".nivel_benzina95 / 2.0;
   "Bazine"."motorina_1/2" := "Bazine".nivel_motorina / 2.0;
   "Bazine"."motorina_premium_1/2" := "Bazine".nivel_motorina_premium / 2.0;
END_REGION

REGION Network 14: bazin la jumate
   RUNG wire#powerrail
      { S7_Templates := "SrcType := Real" } LE_Contact(in1 := "Bazine".benzina_90, in2 := "Bazine"."benzina_90_1/2")
      { S7_Templates := "SrcType := Real" } GT_Contact(in1 := "Bazine".benzina_90, in2 := 0.0)
      Coil( "Alarme".alarme_vect[5] )
   END_RUNG
   RUNG wire#powerrail
      { S7_Templates := "SrcType := Real" } LE_Contact(in1 := "Bazine".benzina_95, in2 := "Bazine"."benzina_95_1/2")
      { S7_Templates := "SrcType := Real" } GT_Contact(in1 := "Bazine".benzina_95, in2 := 0.0)
      Coil( "Alarme".alarme_vect[6] )
   END_RUNG
   RUNG wire#powerrail
      { S7_Templates := "SrcType := Real" } LE_Contact(in1 := "Bazine".motorina, in2 := "Bazine"."motorina_1/2")
      { S7_Templates := "SrcType := Real" } GT_Contact(in1 := "Bazine".motorina, in2 := 0.0)
      Coil( "Alarme".alarme_vect[7] )
   END_RUNG
   RUNG wire#powerrail
      { S7_Templates := "SrcType := Real" } LE_Contact(in1 := "Bazine".motorina_premium, in2 := "Bazine"."motorina_premium_1/2")
      { S7_Templates := "SrcType := Real" } GT_Contact(in1 := "Bazine".motorina_premium, in2 := 0.0)
      Coil( "Alarme".alarme_vect[8] )
   END_RUNG
   // the same network as SCL:
   "Alarme".alarme_vect[5] := ("Bazine".benzina_90 <= "Bazine"."benzina_90_1/2") AND ("Bazine".benzina_90 > 0.0);
   "Alarme".alarme_vect[6] := ("Bazine".benzina_95 <= "Bazine"."benzina_95_1/2") AND ("Bazine".benzina_95 > 0.0);
   "Alarme".alarme_vect[7] := ("Bazine".motorina <= "Bazine"."motorina_1/2") AND ("Bazine".motorina > 0.0);
   "Alarme".alarme_vect[8] := ("Bazine".motorina_premium <= "Bazine"."motorina_premium_1/2") AND ("Bazine".motorina_premium > 0.0);
END_REGION

REGION Network 15: bazin gol
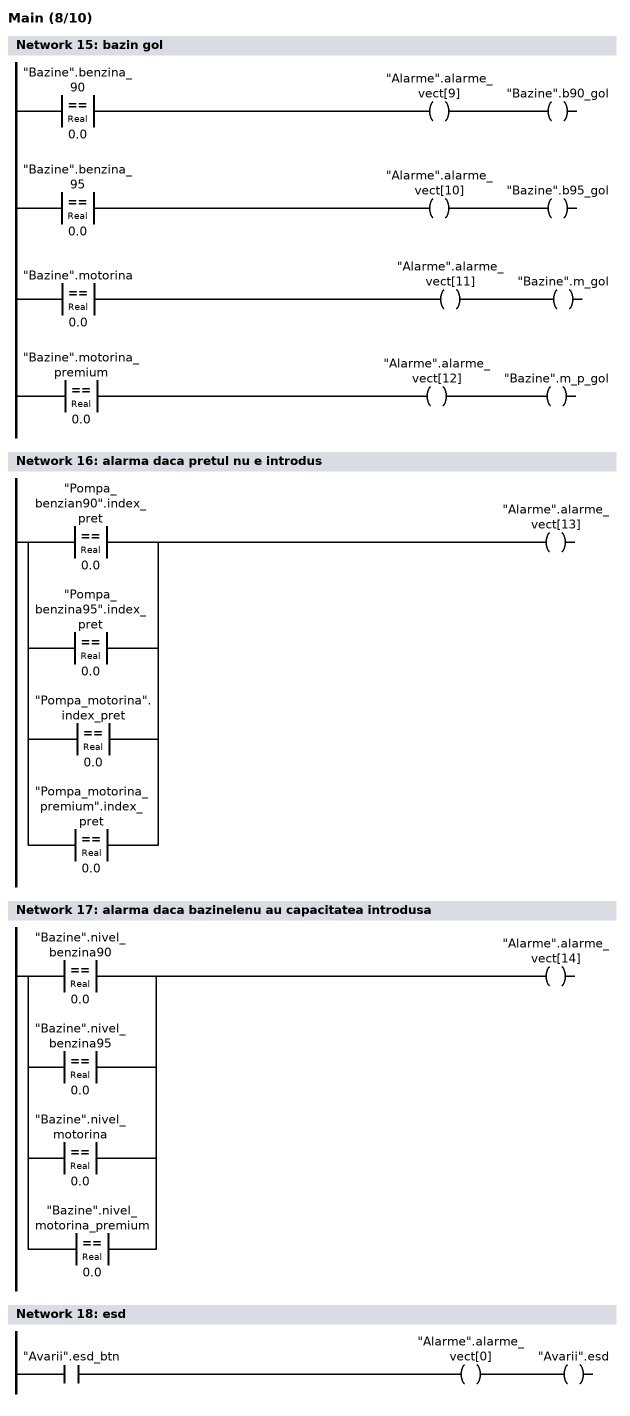
   RUNG wire#powerrail
      { S7_Templates := "SrcType := Real" } EQ_Contact(in1 := "Bazine".benzina_90, in2 := 0.0)
      Coil( "Alarme".alarme_vect[9] )
      Coil( "Bazine".b90_gol )
   END_RUNG
   RUNG wire#powerrail
      { S7_Templates := "SrcType := Real" } EQ_Contact(in1 := "Bazine".benzina_95, in2 := 0.0)
      Coil( "Alarme".alarme_vect[10] )
      Coil( "Bazine".b95_gol )
   END_RUNG
   RUNG wire#powerrail
      { S7_Templates := "SrcType := Real" } EQ_Contact(in1 := "Bazine".motorina, in2 := 0.0)
      Coil( "Alarme".alarme_vect[11] )
      Coil( "Bazine".m_gol )
   END_RUNG
   RUNG wire#powerrail
      { S7_Templates := "SrcType := Real" } EQ_Contact(in1 := "Bazine".motorina_premium, in2 := 0.0)
      Coil( "Alarme".alarme_vect[12] )
      Coil( "Bazine".m_p_gol )
   END_RUNG
   // the same network as SCL:
   "Alarme".alarme_vect[9] := "Bazine".benzina_90 = 0.0;
   "Bazine".b90_gol := "Bazine".benzina_90 = 0.0;
   "Alarme".alarme_vect[10] := "Bazine".benzina_95 = 0.0;
   "Bazine".b95_gol := "Bazine".benzina_95 = 0.0;
   "Alarme".alarme_vect[11] := "Bazine".motorina = 0.0;
   "Bazine".m_gol := "Bazine".motorina = 0.0;
   "Alarme".alarme_vect[12] := "Bazine".motorina_premium = 0.0;
   "Bazine".m_p_gol := "Bazine".motorina_premium = 0.0;
END_REGION

REGION Network 16: alarma daca pretul nu e introdus
   RUNG wire#powerrail
      { S7_Templates := "SrcType := Real" } EQ_Contact(in1 := "Pompa_benzian90".index_pret, in2 := 0.0)
      wire#w1
      Coil( "Alarme".alarme_vect[13] )
   END_RUNG
   RUNG wire#powerrail
      { S7_Templates := "SrcType := Real" } EQ_Contact(in1 := "Pompa_benzina95".index_pret, in2 := 0.0)
   END_RUNG wire#w1
   RUNG wire#powerrail
      { S7_Templates := "SrcType := Real" } EQ_Contact(in1 := "Pompa_motorina".index_pret, in2 := 0.0)
   END_RUNG wire#w1
   RUNG wire#powerrail
      { S7_Templates := "SrcType := Real" } EQ_Contact(in1 := "Pompa_motorina_premium".index_pret, in2 := 0.0)
   END_RUNG wire#w1
   // the same network as SCL:
   "Alarme".alarme_vect[13] := ("Pompa_benzian90".index_pret = 0.0) OR ("Pompa_benzina95".index_pret = 0.0) OR ("Pompa_motorina".index_pret = 0.0) OR ("Pompa_motorina_premium".index_pret = 0.0);
END_REGION

REGION Network 17: alarma daca bazinelenu au capacitatea introdusa
   RUNG wire#powerrail
      { S7_Templates := "SrcType := Real" } EQ_Contact(in1 := "Bazine".nivel_benzina90, in2 := 0.0)
      wire#w1
      Coil( "Alarme".alarme_vect[14] )
   END_RUNG
   RUNG wire#powerrail
      { S7_Templates := "SrcType := Real" } EQ_Contact(in1 := "Bazine".nivel_benzina95, in2 := 0.0)
   END_RUNG wire#w1
   RUNG wire#powerrail
      { S7_Templates := "SrcType := Real" } EQ_Contact(in1 := "Bazine".nivel_motorina, in2 := 0.0)
   END_RUNG wire#w1
   RUNG wire#powerrail
      { S7_Templates := "SrcType := Real" } EQ_Contact(in1 := "Bazine".nivel_motorina_premium, in2 := 0.0)
   END_RUNG wire#w1
   // the same network as SCL:
   "Alarme".alarme_vect[14] := ("Bazine".nivel_benzina90 = 0.0) OR ("Bazine".nivel_benzina95 = 0.0) OR ("Bazine".nivel_motorina = 0.0) OR ("Bazine".nivel_motorina_premium = 0.0);
END_REGION

REGION Network 18: esd
   RUNG wire#powerrail
      Contact( "Avarii".esd_btn )
      Coil( "Alarme".alarme_vect[0] )
      Coil( "Avarii".esd )
   END_RUNG
   // the same network as SCL:
   "Alarme".alarme_vect[0] := "Avarii".esd_btn;
   "Avarii".esd := "Avarii".esd_btn;
END_REGION

REGION Network 19: reset esd
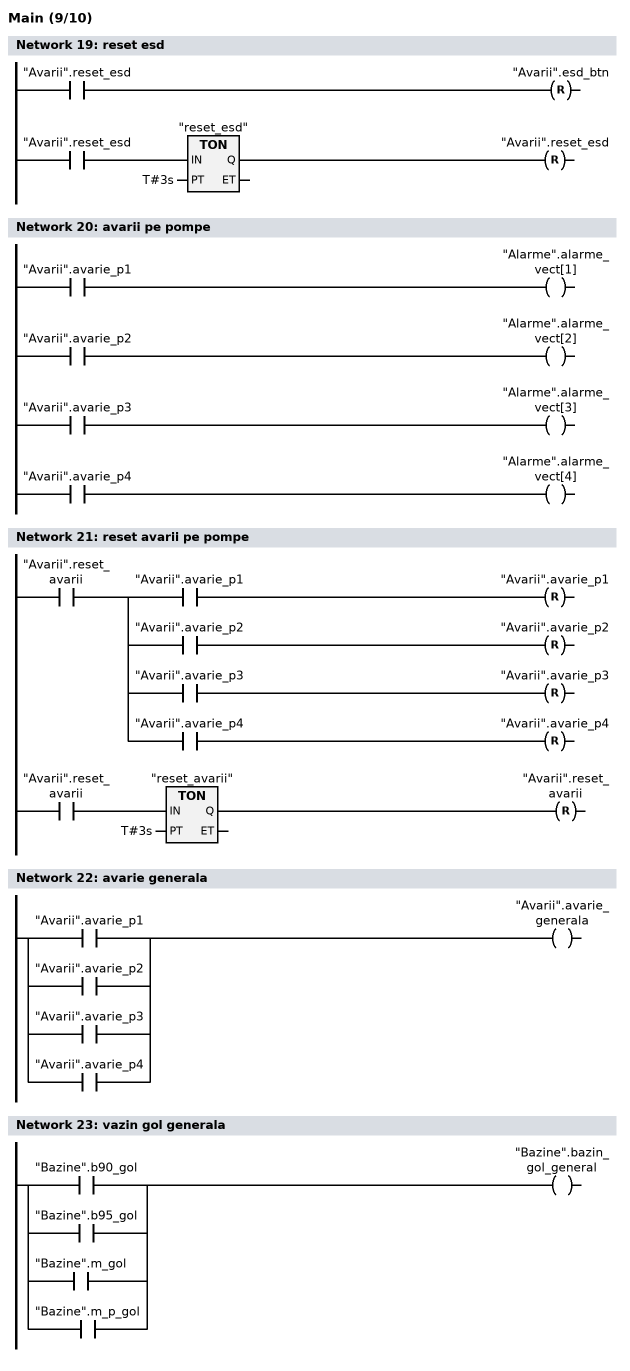
   IF "Avarii".reset_esd THEN "Avarii".esd_btn := FALSE; END_IF;
   "reset_esd".TON(IN := "Avarii".reset_esd, PT := T#3s);
   IF "reset_esd".Q THEN "Avarii".reset_esd := FALSE; END_IF;
END_REGION

REGION Network 20: avarii pe pompe
   RUNG wire#powerrail
      Contact( "Avarii".avarie_p1 )
      Coil( "Alarme".alarme_vect[1] )
   END_RUNG
   RUNG wire#powerrail
      Contact( "Avarii".avarie_p2 )
      Coil( "Alarme".alarme_vect[2] )
   END_RUNG
   RUNG wire#powerrail
      Contact( "Avarii".avarie_p3 )
      Coil( "Alarme".alarme_vect[3] )
   END_RUNG
   RUNG wire#powerrail
      Contact( "Avarii".avarie_p4 )
      Coil( "Alarme".alarme_vect[4] )
   END_RUNG
   // the same network as SCL:
   "Alarme".alarme_vect[1] := "Avarii".avarie_p1;
   "Alarme".alarme_vect[2] := "Avarii".avarie_p2;
   "Alarme".alarme_vect[3] := "Avarii".avarie_p3;
   "Alarme".alarme_vect[4] := "Avarii".avarie_p4;
END_REGION

REGION Network 21: reset avarii pe pompe
   IF "Avarii".reset_avarii AND "Avarii".avarie_p1 THEN "Avarii".avarie_p1 := FALSE; END_IF;
   IF "Avarii".reset_avarii AND "Avarii".avarie_p2 THEN "Avarii".avarie_p2 := FALSE; END_IF;
   IF "Avarii".reset_avarii AND "Avarii".avarie_p3 THEN "Avarii".avarie_p3 := FALSE; END_IF;
   IF "Avarii".reset_avarii AND "Avarii".avarie_p4 THEN "Avarii".avarie_p4 := FALSE; END_IF;
   "reset_avarii".TON(IN := "Avarii".reset_avarii, PT := T#3s);
   IF "reset_avarii".Q THEN "Avarii".reset_avarii := FALSE; END_IF;
END_REGION

REGION Network 22: avarie generala
   RUNG wire#powerrail
      Contact( "Avarii".avarie_p1 )
      wire#w1
      Coil( "Avarii".avarie_generala )
   END_RUNG
   RUNG wire#powerrail
      Contact( "Avarii".avarie_p2 )
   END_RUNG wire#w1
   RUNG wire#powerrail
      Contact( "Avarii".avarie_p3 )
   END_RUNG wire#w1
   RUNG wire#powerrail
      Contact( "Avarii".avarie_p4 )
   END_RUNG wire#w1
   // the same network as SCL:
   "Avarii".avarie_generala := "Avarii".avarie_p1 OR "Avarii".avarie_p2 OR "Avarii".avarie_p3 OR "Avarii".avarie_p4;
END_REGION

REGION Network 23: vazin gol generala
   RUNG wire#powerrail
      Contact( "Bazine".b90_gol )
      wire#w1
      Coil( "Bazine".bazin_gol_general )
   END_RUNG
   RUNG wire#powerrail
      Contact( "Bazine".b95_gol )
   END_RUNG wire#w1
   RUNG wire#powerrail
      Contact( "Bazine".m_gol )
   END_RUNG wire#w1
   RUNG wire#powerrail
      Contact( "Bazine".m_p_gol )
   END_RUNG wire#w1
   // the same network as SCL:
   "Bazine".bazin_gol_general := "Bazine".b90_gol OR "Bazine".b95_gol OR "Bazine".m_gol OR "Bazine".m_p_gol;
END_REGION

REGION Network 24: plata generala
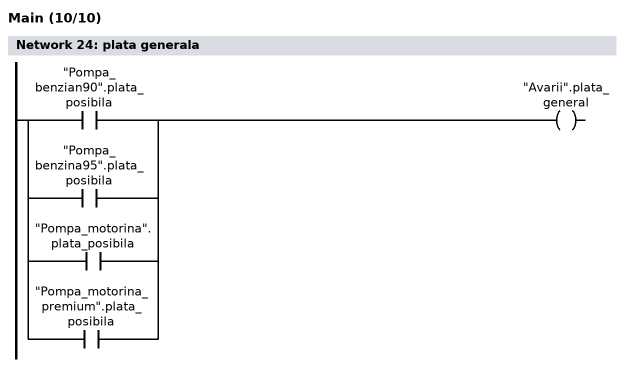
   RUNG wire#powerrail
      Contact( "Pompa_benzian90".plata_posibila )
      wire#w1
      Coil( "Avarii".plata_general )
   END_RUNG
   RUNG wire#powerrail
      Contact( "Pompa_benzina95".plata_posibila )
   END_RUNG wire#w1
   RUNG wire#powerrail
      Contact( "Pompa_motorina".plata_posibila )
   END_RUNG wire#w1
   RUNG wire#powerrail
      Contact( "Pompa_motorina_premium".plata_posibila )
   END_RUNG wire#w1
   // the same network as SCL:
   "Avarii".plata_general := "Pompa_benzian90".plata_posibila OR "Pompa_benzina95".plata_posibila OR "Pompa_motorina".plata_posibila OR "Pompa_motorina_premium".plata_posibila;
END_REGION
END_ORGANIZATION_BLOCK

(* ===== HMI "HMI_RT_1" =====
system functions are stored by id; their names below are inferred from use
connection "HMI_Connection_1": ETHERNET, SMART_S7_1500_OMS

HMI tags "Default tag table"
   "Tag_ScreenNumber" : UInt, internal
   "Alarme_alarme_gather" : Word = PLC Alarme.alarme_gather, 1 s
   "Bazine_benzina_90" : Real = PLC Bazine.benzina_90, 1 s
   "Bazine_benzina_95" : Real = PLC Bazine.benzina_95, 1 s
   "Bazine_motorina" : Real = PLC Bazine.motorina, 1 s
   "Bazine_motorina_premium" : Real = PLC Bazine.motorina_premium, 1 s
   "Butoane_umplere_bazine_btn_b90" : Bool = PLC Butoane_umplere_bazine.btn_b90, 1 s
   "Butoane_umplere_bazine_btn_b95" : Bool = PLC Butoane_umplere_bazine.btn_b95, 1 s
   "Butoane_umplere_bazine_btn_m" : Bool = PLC Butoane_umplere_bazine.btn_m, 1 s
   "Butoane_umplere_bazine_btn_m_p" : Bool = PLC Butoane_umplere_bazine.btn_m_p, 1 s
   "Avarii_esd" : Bool = PLC Avarii.esd, 1 s
   "Avarii_esd_btn" : Bool = PLC Avarii.esd_btn, 1 s
   "Avarii_reset_esd" : Bool = PLC Avarii.reset_esd, 1 s
   "Avarii_avarie_p1" : Bool = PLC Avarii.avarie_p1, 1 s
   "Avarii_avarie_p2" : Bool = PLC Avarii.avarie_p2, 1 s
   "Avarii_avarie_p3" : Bool = PLC Avarii.avarie_p3, 1 s
   "Avarii_avarie_p4" : Bool = PLC Avarii.avarie_p4, 1 s
   "Avarii_reset_avarii" : Bool = PLC Avarii.reset_avarii, 1 s
   "Bazine_nivel_benzina90" : Real = PLC Bazine.nivel_benzina90, 1 s
   "Bazine_nivel_benzina95" : Real = PLC Bazine.nivel_benzina95, 1 s
   "Bazine_nivel_motorina" : Real = PLC Bazine.nivel_motorina, 1 s
   "Bazine_nivel_motorina_premium" : Real = PLC Bazine.nivel_motorina_premium, 1 s
   "Pompa_benzian90_index_pret" : Real = PLC Pompa_benzian90.index_pret, 1 s
   "Pompa_benzina95_index_pret" : Real = PLC Pompa_benzina95.index_pret, 1 s
   "Pompa_motorina_index_pret" : Real = PLC Pompa_motorina.index_pret, 1 s
   "Pompa_motorina_premium_index_pret" : Real = PLC Pompa_motorina_premium.index_pret, 1 s
   "Pompa_benzian90_blocare" : Bool = PLC Pompa_benzian90.blocare, 1 s
   "Pompa_benzian90_permisiune_pompa" : Bool = PLC Pompa_benzian90.permisiune_pompa, 1 s
   "Pompa_benzian90_plata_posibila" : Bool = PLC Pompa_benzian90.plata_posibila, 1 s
   "Pompa_benzian90_permisiune_start" : Bool = PLC Pompa_benzian90.permisiune_start, 1 s
   "Pompa_benzian90_cantitate" : Real = PLC Pompa_benzian90.cantitate, 1 s
   "Pompa_benzian90_pret" : Real = PLC Pompa_benzian90.pret, 1 s
   "Pompa_benzian90_scoasa" : Bool = PLC Pompa_benzian90.scoasa, 1 s
   "Pompa_benzian90_pune_inapoi" : Bool = PLC Pompa_benzian90.pune_inapoi, 1 s
   "Pompa_benzian90_start_clapeta" : Bool = PLC Pompa_benzian90.start_clapeta, 1 s
   "Pompa_benzian90_buton_plata" : Bool = PLC Pompa_benzian90.buton_plata, 1 s
   "Pompa_benzian90_nivel_pompa" : Real = PLC Pompa_benzian90.nivel_pompa, 1 s
   "Pompa_benzina95_nivel_pompa" : Real = PLC Pompa_benzina95.nivel_pompa, 1 s
   "Pompa_motorina_nivel_pompa" : Real = PLC Pompa_motorina.nivel_pompa, 1 s
   "Pompa_motorina_premium_nivel_pompa" : Real = PLC Pompa_motorina_premium.nivel_pompa, 1 s
   "Pompa_benzina95_blocare" : Bool = PLC Pompa_benzina95.blocare, 1 s
   "Pompa_benzina95_permisiune_pompa" : Bool = PLC Pompa_benzina95.permisiune_pompa, 1 s
   "Pompa_benzina95_permisiune_start" : Bool = PLC Pompa_benzina95.permisiune_start, 1 s
   "Pompa_benzina95_plata_posibila" : Bool = PLC Pompa_benzina95.plata_posibila, 1 s
   "Pompa_benzina95_pret" : Real = PLC Pompa_benzina95.pret, 1 s
   "Pompa_benzina95_cantitate" : Real = PLC Pompa_benzina95.cantitate, 1 s
   "Pompa_benzina95_scoasa" : Bool = PLC Pompa_benzina95.scoasa, 1 s
   "Pompa_benzina95_start_clapeta" : Bool = PLC Pompa_benzina95.start_clapeta, 1 s
   "Pompa_motorina_blocare" : Bool = PLC Pompa_motorina.blocare, 1 s
   "Pompa_motorina_permisiune_pompa" : Bool = PLC Pompa_motorina.permisiune_pompa, 1 s
   "Pompa_motorina_plata_posibila" : Bool = PLC Pompa_motorina.plata_posibila, 1 s
   "Pompa_motorina_permisiune_start" : Bool = PLC Pompa_motorina.permisiune_start, 1 s
   "Pompa_motorina_scoasa" : Bool = PLC Pompa_motorina.scoasa, 1 s
   "Pompa_motorina_start_clapeta" : Bool = PLC Pompa_motorina.start_clapeta, 1 s
   "Pompa_motorina_cantitate" : Real = PLC Pompa_motorina.cantitate, 1 s
   "Pompa_motorina_pret" : Real = PLC Pompa_motorina.pret, 1 s
   "Pompa_motorina_buton_plata" : Bool = PLC Pompa_motorina.buton_plata, 1 s
   "Pompa_motorina_premium_buton_plata" : Bool = PLC Pompa_motorina_premium.buton_plata, 1 s
   "Pompa_benzina95_buton_plata" : Bool = PLC Pompa_benzina95.buton_plata, 1 s
   "Pompa_motorina_premium_cantitate" : Real = PLC Pompa_motorina_premium.cantitate, 1 s
   "Pompa_motorina_premium_pret" : Real = PLC Pompa_motorina_premium.pret, 1 s
   "Pompa_motorina_premium_blocare" : Bool = PLC Pompa_motorina_premium.blocare, 1 s
   "Pompa_motorina_premium_scoasa" : Bool = PLC Pompa_motorina_premium.scoasa, 1 s
   "Pompa_motorina_premium_permisiune_start" : Bool = PLC Pompa_motorina_premium.permisiune_start, 1 s
   "Pompa_motorina_premium_permisiune_pompa" : Bool = PLC Pompa_motorina_premium.permisiune_pompa, 1 s
   "Pompa_motorina_premium_start_clapeta" : Bool = PLC Pompa_motorina_premium.start_clapeta, 1 s
   "Pompa_motorina_premium_led_rosu" : Bool = PLC Pompa_motorina_premium.led_rosu, 1 s
   "Pompa_motorina_led_rosu" : Bool = PLC Pompa_motorina.led_rosu, 1 s
   "Pompa_benzina95_led_rosu" : Bool = PLC Pompa_benzina95.led_rosu, 1 s
   "Pompa_benzian90_led_rosu" : Bool = PLC Pompa_benzian90.led_rosu, 1 s
   "Pompa_motorina_premium_plata_posibila" : Bool = PLC Pompa_motorina_premium.plata_posibila, 1 s

discrete alarms
   1: 'ESD', class Errors, trigger "Alarme_alarme_gather" bit 0
   2: 'Avarie pompa 1', class Errors, trigger "Alarme_alarme_gather" bit 1
   3: 'Avarie pompa 2', class Errors, trigger "Alarme_alarme_gather" bit 2
   4: 'Avarie pompa 3', class Errors, trigger "Alarme_alarme_gather" bit 3
   5: 'Avarie pompa 4', class Errors, trigger "Alarme_alarme_gather" bit 4
   6: 'Bazin benzina90 la jumatate', class Errors, trigger "Alarme_alarme_gather" bit 5
   7: 'Bazin benzina95 la jumatate', class Errors, trigger "Alarme_alarme_gather" bit 6
   8: 'Bazin motorina la jumatate', class Errors, trigger "Alarme_alarme_gather" bit 7
   9: 'Bazin motorina premium la jumatate', class Errors, trigger "Alarme_alarme_gather" bit 8
   10: 'Bazin benzina90 gol', class Errors, trigger "Alarme_alarme_gather" bit 9
   11: 'Bazin benzina95 gol', class Errors, trigger "Alarme_alarme_gather" bit 10
   12: 'Bazin motorina gol', class Errors, trigger "Alarme_alarme_gather" bit 11
   13: 'Bazin motorina premium gol', class Errors, trigger "Alarme_alarme_gather" bit 12
   14: 'Preturi neinregistrate', class Errors, trigger "Alarme_alarme_gather" bit 13
   15: 'Niveluri bazine neintregistrate', class Errors, trigger "Alarme_alarme_gather" bit 14
   16: 'Nivele bazine nesetate', class Errors, trigger "Alarme_alarme_gather" bit 15

Template "Template_1" 800x480
   Button "Exit" at 722,440 size 55x39; TextOff 'Exit'; PictureOff "ExitRuntime_KTP900_Basic_PN_TR"; PictureOn "ExitRuntime_KTP900_Basic_PN_TR"
      on Release: StopRuntime(0)
   Button "Template_Button" at 622,440 size 55x39; TextOff 'Text'
   Button "Template_Button_1" at 522,440 size 55x39; TextOff 'Text'
   Button "Alarms" at 622,440 size 55x39; TextOff 'Alarms'; PictureOff "AlarmDisplay_KTP900_Basic_PN_TR"; PictureOn "AlarmDisplay_KTP900_Basic_PN_TR"
      on Release: function_ef3f5d25("Alarm window_1", -1)
   Button "Start screen" at 522,440 size 55x39; TextOff 'Start screen'; PictureOff "NavigateHome_KTP900_Basic_PN_TR"; PictureOn "NavigateHome_KTP900_Basic_PN_TR"
      on Release: ActivateScreen("Main", 0)

screen "Main" 800x480, template "Template_1"
   on GenerateScreen: SetTag("Tag_ScreenNumber", 1)
   TextField "Template_Text field_1" at 34,456 size 35x20; Text 'Main'
   TextField "Template_Text field_2" at 122,455 size 60x20; Text 'Simulare'
   TextField "Template_Text field_3" at 228,455 size 47x20; Text 'Bazine'
   TextField "Text field_2" at 367,10 size 51x27; Text 'Main'
   TextField "Text field_1" at 680,71 size 50x22; Text 'Avarii'
   Button "Button_1" at 680,117 size 96x32; TextOff 'Pompa1'
      on Click: SetBit("Avarii_avarie_p1")
   Circle "Circle_1" at 629,114 size 37x37
      Appearance <- "Avarii_avarie_p1"
   Button "Button_2" at 680,174 size 96x32; TextOff 'Pompa2'
      on Click: SetBit("Avarii_avarie_p2")
   Circle "Circle_2" at 629,171 size 37x37
      Appearance <- "Avarii_avarie_p2"
   Button "Button_3" at 680,231 size 96x32; TextOff 'Pompa3'
      on Click: SetBit("Avarii_avarie_p3")
   Circle "Circle_3" at 629,228 size 37x37
      Appearance <- "Avarii_avarie_p3"
   Button "Button_4" at 680,288 size 96x32; TextOff 'Pompa4'
      on Click: SetBit("Avarii_avarie_p4")
   Circle "Circle_4" at 629,285 size 37x37
      Appearance <- "Avarii_avarie_p4"
   Button "Button_5" at 657,348 size 96x32; TextOff 'Reset'
      on Click: SetBit("Avarii_reset_avarii")
   Circle "Circle_5" at 432,306 size 48x48
      Appearance <- "Avarii_esd"
   Button "Button_6" at 428,363 size 58x32; TextOff 'ESD'
      on Click: SetBit("Avarii_esd_btn")
   Button "Button_7" at 428,401 size 58x32; TextOff 'RESET'
      on Click: SetBit("Avarii_reset_esd")
   TextField "Text field_3" at 126,84 size 51x22; Text 'Setari'
   TextField "Text field_4" at 9,162 size 60x20; Text 'Pompa 1'
   IOField "I/O field_1" at 96,158 size 96x32; FormatPattern 9999; Unit L
      ProcessValue <- "Bazine_nivel_benzina90"
   IOField "I/O field_2" at 210,158 size 96x32; FormatPattern 9.99; Unit RON
      ProcessValue <- "Pompa_benzian90_index_pret"
   TextField "Text field_5" at 119,125 size 39x20; Text 'Bazin'
   TextField "Text field_6" at 237,124 size 33x20; Text 'Pret'
   TextField "Text field_7" at 9,209 size 60x20; Text 'Pompa 2'
   IOField "I/O field_3" at 96,205 size 96x32; FormatPattern 9999; Unit L
      ProcessValue <- "Bazine_nivel_benzina95"
   IOField "I/O field_4" at 210,205 size 96x32; FormatPattern 9.99; Unit RON
      ProcessValue <- "Pompa_benzina95_index_pret"
   TextField "Text field_8" at 9,256 size 60x20; Text 'Pompa 3'
   IOField "I/O field_5" at 96,252 size 96x32; FormatPattern 9999; Unit L
      ProcessValue <- "Bazine_nivel_motorina"
   IOField "I/O field_6" at 210,252 size 96x32; FormatPattern 9.99; Unit RON
      ProcessValue <- "Pompa_motorina_index_pret"
   TextField "Text field_9" at 9,303 size 60x20; Text 'Pompa 4'
   IOField "I/O field_7" at 96,299 size 96x32; FormatPattern 9999; Unit L
      ProcessValue <- "Bazine_nivel_motorina_premium"
   IOField "I/O field_8" at 210,299 size 96x32; FormatPattern 9.99; Unit RON
      ProcessValue <- "Pompa_motorina_premium_index_pret"

screen "Simulare" 800x480
   TextField "Template_Text field_1" at 34,456 size 35x20; Text 'Main'
   TextField "Template_Text field_2" at 122,455 size 60x20; Text 'Simulare'
   TextField "Template_Text field_3" at 228,455 size 47x20; Text 'Bazine'
   TextField "Text field_2" at 365,10 size 89x27; Text 'Simulare'
   Rectangle "Rectangle_1" at 77,177 size 51x180
      Appearance <- "Pompa_benzian90_permisiune_start"
   Circle "Circle_1" at 53,94 size 36x36
      Appearance <- "Pompa_benzian90_blocare"
   Circle "Circle_2" at 117,94 size 36x36
      Appearance <- "Pompa_benzian90_permisiune_pompa"
   TextField "Text field_1" at 69,144 size 71x20; Text 'Benzina90'
   TextField "Text field_3" at 50,72 size 45x20; Text 'Blocat'
   TextField "Text field_4" at 113,72 size 48x20; Text 'Pompa'
   IOField "I/O field_1" at 2,194 size 55x32; FormatPattern 9.99
      ProcessValue <- "Pompa_benzian90_index_pret"
   TextField "Text field_5" at 4,169 size 48x20; Text 'Pret/L'
   IOField "I/O field_2" at 1,254 size 55x32; FormatPattern 999
      ProcessValue <- "Pompa_benzian90_cantitate"
   TextField "Text field_6" at 3,229 size 66x20; Text 'Cantitate'
   IOField "I/O field_3" at 0,314 size 61x32; FormatPattern 999.99
      ProcessValue <- "Pompa_benzian90_pret"
   TextField "Text field_7" at 2,289 size 68x20; Text 'Pret total'
   Circle "Circle_3" at 149,171 size 32x32
      Visibility <- "Pompa_benzian90_plata_posibila"
      Appearance <- "Pompa_benzian90_led_rosu"
   Button "Button_1" at 142,212 size 48x25; TextOff 'Plata'
      Visibility <- "Pompa_benzian90_plata_posibila"
      on Click: SetBit("Pompa_benzian90_buton_plata")
   Button "Button_2" at 40,377 size 55x26; TextOff 'Scoate'
      Visibility <- "Pompa_benzian90_scoasa"
      on Click: SetTag("Pompa_benzian90_scoasa", 1)
   Button "Button_3" at 105,410 size 55x26; TextOff 'Stop'
      Visibility <- "Pompa_benzian90_start_clapeta"
      on Click: SetTag("Pompa_benzian90_start_clapeta", 0)
   Button "Button_4" at 105,376 size 55x26; TextOff 'Inapoi'
      Visibility <- "Pompa_benzian90_pune_inapoi"
      on Click: SetTag("Pompa_benzian90_scoasa", 0)
   Button "Button_5" at 40,410 size 55x26; TextOff 'Start'
      Visibility <- "Pompa_benzian90_start_clapeta"
      on Click: SetTag("Pompa_benzian90_start_clapeta", 1)
   Rectangle "Rectangle_2" at 283,172 size 51x180
      Appearance <- "Pompa_benzina95_permisiune_start"
   Circle "Circle_4" at 259,89 size 36x36
      Appearance <- "Pompa_benzina95_blocare"
   Circle "Circle_5" at 323,89 size 36x36
      Appearance <- "Pompa_benzina95_permisiune_pompa"
   TextField "Text field_8" at 277,144 size 71x20; Text 'Benzina95'
   TextField "Text field_9" at 256,67 size 45x20; Text 'Blocat'
   TextField "Text field_10" at 319,67 size 48x20; Text 'Pompa'
   IOField "I/O field_4" at 212,194 size 55x32; FormatPattern 9.99
      ProcessValue <- "Pompa_benzina95_index_pret"
   TextField "Text field_11" at 214,169 size 48x20; Text 'Pret/L'
   IOField "I/O field_5" at 211,254 size 55x32; FormatPattern 999
      ProcessValue <- "Pompa_benzina95_cantitate"
   TextField "Text field_12" at 213,229 size 66x20; Text 'Cantitate'
   IOField "I/O field_6" at 210,314 size 61x32; FormatPattern 999.99
      ProcessValue <- "Pompa_benzina95_pret"
   TextField "Text field_13" at 212,289 size 68x20; Text 'Pret total'
   Circle "Circle_6" at 356,171 size 32x32
      Visibility <- "Pompa_benzina95_plata_posibila"
      Appearance <- "Pompa_benzina95_led_rosu"
   Button "Button_6" at 349,212 size 48x25; TextOff 'Plata'
      Visibility <- "Pompa_benzina95_plata_posibila"
      on Click: SetBit("Pompa_benzina95_buton_plata")
   Button "Button_7" at 247,377 size 55x26; TextOff 'Scoate'
      on Click: SetTag("Pompa_benzina95_scoasa", 1)
      Visibility <- "Pompa_benzina95_scoasa"
   Button "Button_8" at 312,410 size 55x26; TextOff 'Stop'
      on Click: SetTag("Pompa_benzina95_start_clapeta", 0)
      Visibility <- "Pompa_benzina95_start_clapeta"
   Button "Button_9" at 312,376 size 55x26; TextOff 'Inapoi'
      on Click: SetTag("Pompa_benzina95_scoasa", 0)
      Visibility <- "Pompa_benzina95_scoasa"
   Button "Button_10" at 247,410 size 55x26; TextOff 'Start'
      on Click: SetTag("Pompa_benzina95_start_clapeta", 1)
      Visibility <- "Pompa_benzina95_start_clapeta"
   Rectangle "Rectangle_4" at 487,177 size 51x180
      Appearance <- "Pompa_motorina_permisiune_start"
   Circle "Circle_7" at 463,94 size 36x36
      Appearance <- "Pompa_motorina_blocare"
   Circle "Circle_8" at 527,94 size 36x36
      Appearance <- "Pompa_motorina_permisiune_pompa"
   TextField "Text field_14" at 481,144 size 63x20; Text 'Motorina'
   TextField "Text field_15" at 460,72 size 45x20; Text 'Blocat'
   TextField "Text field_16" at 523,72 size 48x20; Text 'Pompa'
   IOField "I/O field_7" at 419,194 size 55x32; FormatPattern 9.99
      ProcessValue <- "Pompa_motorina_index_pret"
   TextField "Text field_17" at 421,169 size 48x20; Text 'Pret/L'
   IOField "I/O field_8" at 418,254 size 55x32; FormatPattern 999
      ProcessValue <- "Pompa_motorina_cantitate"
   TextField "Text field_18" at 420,229 size 66x20; Text 'Cantitate'
   IOField "I/O field_9" at 417,314 size 62x32; FormatPattern 999.99
      ProcessValue <- "Pompa_motorina_pret"
   TextField "Text field_19" at 419,289 size 68x20; Text 'Pret total'
   Circle "Circle_9" at 559,171 size 32x32
      Appearance <- "Pompa_motorina_led_rosu"
      Visibility <- "Pompa_motorina_plata_posibila"
   Button "Button_11" at 552,212 size 48x25; TextOff 'Plata'
      Visibility <- "Pompa_motorina_plata_posibila"
      on Click: SetBit("Pompa_motorina_buton_plata")
   Button "Button_12" at 450,377 size 55x26; TextOff 'Scoate'
      on Click: SetTag("Pompa_motorina_scoasa", 1)
      Visibility <- "Pompa_motorina_scoasa"
   Button "Button_13" at 515,410 size 55x26; TextOff 'Stop'
      on Click: SetTag("Pompa_motorina_start_clapeta", 0)
      Visibility <- "Pompa_motorina_start_clapeta"
   Button "Button_14" at 515,376 size 55x26; TextOff 'Inapoi'
      on Click: SetTag("Pompa_motorina_scoasa", 0)
      Visibility <- "Pompa_motorina_scoasa"
   Button "Button_15" at 450,410 size 55x26; TextOff 'Start'
      on Click: SetTag("Pompa_motorina_start_clapeta", 1)
      Visibility <- "Pompa_motorina_start_clapeta"
   Rectangle "Rectangle_5" at 687,177 size 51x180
      Appearance <- "Pompa_motorina_premium_permisiune_start"
   Circle "Circle_10" at 663,94 size 36x36
      Appearance <- "Pompa_motorina_premium_blocare"
   Circle "Circle_11" at 727,94 size 36x36
      Appearance <- "Pompa_motorina_premium_permisiune_pompa"
   TextField "Text field_20" at 653,144 size 122x20; Text 'Motorina premium'
   TextField "Text field_21" at 660,72 size 45x20; Text 'Blocat'
   TextField "Text field_22" at 723,72 size 48x20; Text 'Pompa'
   IOField "I/O field_10" at 620,194 size 55x32; FormatPattern 9.99
      ProcessValue <- "Pompa_motorina_premium_index_pret"
   TextField "Text field_23" at 622,169 size 48x20; Text 'Pret/L'
   IOField "I/O field_11" at 619,254 size 55x32; FormatPattern 999
      ProcessValue <- "Pompa_motorina_premium_cantitate"
   TextField "Text field_24" at 621,229 size 66x20; Text 'Cantitate'
   IOField "I/O field_12" at 618,314 size 61x32; FormatPattern 999.99
      ProcessValue <- "Pompa_motorina_premium_pret"
   TextField "Text field_25" at 620,289 size 68x20; Text 'Pret total'
   Circle "Circle_12" at 756,171 size 32x32
      Appearance <- "Pompa_motorina_premium_led_rosu"
      Visibility <- "Pompa_motorina_premium_plata_posibila"
   Button "Button_16" at 749,212 size 48x25; TextOff 'Plata'
      on Click: SetBit("Pompa_motorina_premium_buton_plata")
      Visibility <- "Pompa_motorina_premium_plata_posibila"
   Button "Button_17" at 650,377 size 55x26; TextOff 'Scoate'
      on Click: SetTag("Pompa_motorina_premium_scoasa", 1)
      Visibility <- "Pompa_motorina_premium_scoasa"
   Button "Button_18" at 715,410 size 55x26; TextOff 'Stop'
      on Click: SetTag("Pompa_motorina_premium_start_clapeta", 0)
      Visibility <- "Pompa_motorina_premium_start_clapeta"
   Button "Button_19" at 715,376 size 55x26; TextOff 'Inapoi'
      on Click: SetTag("Pompa_motorina_premium_scoasa", 0)
      Visibility <- "Pompa_motorina_premium_scoasa"
   Button "Button_20" at 650,410 size 55x26; TextOff 'Start'
      on Click: SetTag("Pompa_motorina_premium_start_clapeta", 1)
      Visibility <- "Pompa_motorina_premium_start_clapeta"
   IOField "I/O field_13" at 116,45 size 41x24; FormatPattern 99.9
      ProcessValue <- "Pompa_benzian90_nivel_pompa"
   IOField "I/O field_14" at 321,45 size 42x24; FormatPattern 99.9
      ProcessValue <- "Pompa_benzina95_nivel_pompa"
   IOField "I/O field_15" at 524,45 size 41x24; FormatPattern 99.9
      ProcessValue <- "Pompa_motorina_nivel_pompa"
   IOField "I/O field_16" at 726,45 size 41x24; FormatPattern 99.9
      ProcessValue <- "Pompa_motorina_premium_nivel_pompa"

screen "Bazine" 800x480
   TextField "Template_Text field_1" at 34,456 size 35x20; Text 'Main'
   TextField "Template_Text field_2" at 122,455 size 60x20; Text 'Simulare'
   TextField "Template_Text field_3" at 228,455 size 47x20; Text 'Bazine'
   Bar "Bar_1" at 83,107 size 130x260; MinimumValue 0; MaximumValue 1000
      ProcessValue <- "Bazine_benzina_90"
   TextField "Text field_1" at 107,34 size 84x22; Text 'Benzina90'
   IOField "I/O field_1" at 100,63 size 96x32; FormatPattern 9999; Unit L
      ProcessValue <- "Bazine_benzina_90"
   Button "Button_1" at 102,384 size 96x32; TextOff 'Umplere'
      on Click: SetBit("Butoane_umplere_bazine_btn_b90")
   TextField "Text field_2" at 367,10 size 68x27; Text 'Bazine'
   Bar "Bar_2" at 237,107 size 130x260; MinimumValue 0; MaximumValue 1000
      ProcessValue <- "Bazine_benzina_95"
   TextField "Text field_3" at 258,34 size 88x22; Text 'Benzina 95'
   IOField "I/O field_2" at 254,63 size 96x32; FormatPattern 9999; Unit L
      ProcessValue <- "Bazine_benzina_95"
   Button "Button_2" at 256,384 size 96x32; TextOff 'Umplere'
      on Click: SetBit("Butoane_umplere_bazine_btn_b95")
   Bar "Bar_3" at 434,107 size 130x260; MinimumValue 0; MaximumValue 1000
      ProcessValue <- "Bazine_motorina"
   TextField "Text field_4" at 463,34 size 72x22; Text 'Motorina'
   IOField "I/O field_3" at 451,63 size 96x32; FormatPattern 9999; Unit L
      ProcessValue <- "Bazine_motorina"
   Button "Button_3" at 453,384 size 96x32; TextOff 'Umplere'
      on Click: SetBit("Butoane_umplere_bazine_btn_m")
   Bar "Bar_4" at 590,107 size 130x260; MinimumValue 0; MaximumValue 1000
      ProcessValue <- "Bazine_motorina_premium"
   TextField "Text field_5" at 588,34 size 141x22; Text 'Motorina premium'
   IOField "I/O field_4" at 607,63 size 96x32; FormatPattern 9999; Unit L
      ProcessValue <- "Bazine_motorina_premium"
   Button "Button_4" at 609,384 size 96x32; TextOff 'Umplere'
      on Click: SetBit("Butoane_umplere_bazine_btn_m_p")
*)